       CALL #"LCP71_B010_BG8011"
       (
         CM_No       := 10174 ,
         Tab       := 1 ,
         SubTab       := 4 ,
         CfgType       := 0 ,
         CfgInvert       := True ,
         InputRaw       := LCP71_B010_BG8011_DI_ChA ,
         SC_Local       := SL_24_P ,
         CM_ALM        := "dbPlcHmiALM".ALM[10174] ,
       );

NETWORK
TITLE = 10175 - LCP71_B010_BG8012 - Door Hopper feeder Door - Safety Contact

       CALL #"LCP71_B010_BG8012"
       (
         CM_No       := 10175 ,
         Tab       := 1 ,
         SubTab       := 4 ,
         CfgType       := 0 ,
         CfgInvert       := True ,
         InputRaw       := LCP71_B010_BG8012_DI_ChA ,
         SC_Local       := SL_24_P ,
         CM_ALM        := "dbPlcHmiALM".ALM[10175] ,
       );

NETWORK
TITLE = 10176 - LCP71_B010_BG8013 - Hopper feeder Life Line  - Safety Contact

       CALL #"LCP71_B010_BG8013"
       (
         CM_No       := 10176 ,
         Tab       := 1 ,
         SubTab       := 4 ,
         CfgType       := 0 ,
         CfgInvert       := True ,
         InputRaw       := LCP71_B010_BG8013_DI_ChA ,
         SC_Local       := SL_24_P ,
         CM_ALM        := "dbPlcHmiALM".ALM[10176] ,
       );

NETWORK
TITLE = 10177 - LCP71_ES01_SF6134 - Emergency Stop  - Hopper Feeder

       CALL #"LCP71_ES01_SF6134"
       (
         CM_No       := 10177 ,
         Tab       := 1 ,
         SubTab       := 4 ,
         CfgType       := 0 ,
         CfgInvert       := True ,
         InputRaw       := LCP71_ES01_SF6134_DI_ChA ,
         SC_Local       := SL_01 ,
         CM_ALM        := "dbPlcHmiALM".ALM[10177] ,
       );

NETWORK
TITLE = 10178 - LCP71_ES01_SF6135 - Emergency Stop  - LCP71

       CALL #"LCP71_ES01_SF6135"
       (
         CM_No       := 10178 ,
         Tab       := 1 ,
         SubTab       := 4 ,
         CfgType       := 0 ,
         CfgInvert       := True ,
         InputRaw       := LCP71_ES01_SF6135_DI_ChA ,
         SC_Local       := SL_01 ,
         CM_ALM        := "dbPlcHmiALM".ALM[10178] ,
       );

NETWORK
TITLE = 10179 - LCP71_DC01_FC1000 - Power Feed Module 24VDC - Status

       CALL #"LCP71_DC01_FC1000"
       (
         CM_No       := 10179 ,
         Tab       := 13 ,
         SubTab       := 5 ,
         CfgType       := 0 ,
         CfgInvert       := True ,
         InputRaw       := LCP71_DC01_FC1000_DI_Sts ,
         SC_Local       := SL_13 ,
         CM_ALM        := "dbPlcHmiALM".ALM[10179] ,
       );

NETWORK
TITLE = 10180 - LCP71_IO_KF1000 - Point IO - EtherNet/IP Adapter

       CALL #"LCP71_IO_KF1000"
       (
         CM_No       := 10180 ,
         Tab       := 13 ,
         SubTab       := 5 ,
         CfgType       := 0 ,
         CfgInvert       := True ,
         InputRaw       :=  ,
         SC_Local       := SL_13 ,
         CM_ALM        := "dbPlcHmiALM".ALM[10180] ,
       );

NETWORK
TITLE = 10181 - LCP71_IO_KF3007 - 24V DC 8-Point Safety Input Module - SDI

       CALL #"LCP71_IO_KF3007"
       (
         CM_No       := 10181 ,
         Tab       := 13 ,
         SubTab       := 5 ,
         CfgType       := 0 ,
         CfgInvert       := True ,
         InputRaw       :=  ,
         SC_Local       := SL_13 ,
         CM_ALM        := "dbPlcHmiALM".ALM[10181] ,
       );

NETWORK
TITLE = 10182 - LCP71_IO_KF3008 - 24V DC 8-Point Safety Input Module - SDI

       CALL #"LCP71_IO_KF3008"
       (
         CM_No       := 10182 ,
         Tab       := 13 ,
         SubTab       := 5 ,
         CfgType       := 0 ,
         CfgInvert       := True ,
         InputRaw       :=  ,
         SC_Local       := SL_13 ,
         CM_ALM        := "dbPlcHmiALM".ALM[10182] ,
       );

NETWORK
TITLE = 10183 - LCP72_B211_BG8211 - Conderser 2 Door - Safety Contact

       CALL #"LCP72_B211_BG8211"
       (
         CM_No       := 10183 ,
         Tab       := 1 ,
         SubTab       := 4 ,
         CfgType       := 0 ,
         CfgInvert       := True ,
         InputRaw       := LCP72_B211_BG8211_DI_ChA ,
         SC_Local       := SL_24_P12 ,
         CM_ALM        := "dbPlcHmiALM".ALM[10183] ,
       );

NETWORK
TITLE = 10184 - LCP72_B311_BG8311 - Conderser 3 Door - Safety Contact

       CALL #"LCP72_B311_BG8311"
       (
         CM_No       := 10184 ,
         Tab       := 1 ,
         SubTab       := 4 ,
         CfgType       := 0 ,
         CfgInvert       := True ,
         InputRaw       := LCP72_B311_BG8311_DI_ChA ,
         SC_Local       := SL_24_P13 ,
         CM_ALM        := "dbPlcHmiALM".ALM[10184] ,
       );

NETWORK
TITLE = 10185 - LCP72_B411_BG8411 - Conderser 4 Door - Safety Contact

       CALL #"LCP72_B411_BG8411"
       (
         CM_No       := 10185 ,
         Tab       := 1 ,
         SubTab       := 4 ,
         CfgType       := 0 ,
         CfgInvert       := True ,
         InputRaw       := LCP72_B411_BG8411_DI_ChA ,
         SC_Local       := SL_24_P14 ,
         CM_ALM        := "dbPlcHmiALM".ALM[10185] ,
       );

NETWORK
TITLE = 10186 - LCP72_B210_KF6210 - Opening Roll 2 Rotation Monitor - Fault

       CALL #"LCP72_B210_KF6210"
       (
         CM_No       := 10186 ,
         Tab       := 24 ,
         SubTab       := 4 ,
         CfgType       := 0 ,
         CfgInvert       := True ,
         InputRaw       := LCP72_B210_KF6210_DI_Flt ,
         SC_Local       := SL_24_P12 ,
         CM_ALM        := "dbPlcHmiALM".ALM[10186] ,
       );

NETWORK
TITLE = 10187 - LCP72_B210_RL4210 - Metering Feeder 2 - Door Lock Open

       CALL #"LCP72_B210_RL4210"
       (
         CM_No       := 10187 ,
         Tab       := 1 ,
         SubTab       := 4 ,
         CfgType       := 0 ,
         CfgInvert       := True ,
         InputRaw       := LCP72_B210_RL4210_DI_ChA ,
         SC_Local       := SL_24_P12 ,
         CM_ALM        := "dbPlcHmiALM".ALM[10187] ,
       );

NETWORK
TITLE = 10188 - LCP72_B310_KF6310 - Opening Roll 3 Rotation Monitor - Fault

       CALL #"LCP72_B310_KF6310"
       (
         CM_No       := 10188 ,
         Tab       := 24 ,
         SubTab       := 5 ,
         CfgType       := 0 ,
         CfgInvert       := True ,
         InputRaw       := LCP72_B310_KF6310_DI_Flt ,
         SC_Local       := SL_24_P13 ,
         CM_ALM        := "dbPlcHmiALM".ALM[10188] ,
       );

NETWORK
TITLE = 10189 - LCP72_B310_RL4310 - Metering Feeder 3 - Door Lock Open

       CALL #"LCP72_B310_RL4310"
       (
         CM_No       := 10189 ,
         Tab       := 1 ,
         SubTab       := 4 ,
         CfgType       := 0 ,
         CfgInvert       := True ,
         InputRaw       := LCP72_B310_RL4310_DI_ChA ,
         SC_Local       := SL_24_P13 ,
         CM_ALM        := "dbPlcHmiALM".ALM[10189] ,
       );

NETWORK
TITLE = 10190 - LCP72_B410_KF6410 - Opening Roll 4 Rotation Monitor - Fault

       CALL #"LCP72_B410_KF6410"
       (
         CM_No       := 10190 ,
         Tab       := 24 ,
         SubTab       := 6 ,
         CfgType       := 0 ,
         CfgInvert       := True ,
         InputRaw       := LCP72_B410_KF6410_DI_Flt ,
         SC_Local       := SL_24_P14 ,
         CM_ALM        := "dbPlcHmiALM".ALM[10190] ,
       );

NETWORK
TITLE = 10191 - LCP72_B410_RL4410 - Metering Feeder 4 - Door Lock Open

       CALL #"LCP72_B410_RL4410"
       (
         CM_No       := 10191 ,
         Tab       := 1 ,
         SubTab       := 4 ,
         CfgType       := 0 ,
         CfgInvert       := True ,
         InputRaw       := LCP72_B410_RL4410_DI_ChA ,
         SC_Local       := SL_24_P14 ,
         CM_ALM        := "dbPlcHmiALM".ALM[10191] ,
       );

NETWORK
TITLE = 10192 - LCP72_B210_QA1201 - Serel 2 DCM - X-Ray Fault

       CALL #"LCP72_B210_QA1201"
       (
         CM_No       := 10192 ,
         Tab       := 24 ,
         SubTab       := 4 ,
         CfgType       := 0 ,
         CfgInvert       := True ,
         InputRaw       := LCP72_B210_QA1201_DI_Flt ,
         SC_Local       := SL_24_S ,
         CM_ALM        := "dbPlcHmiALM".ALM[10192] ,
       );

NETWORK
TITLE = 10193 - LCP72_B310_QA1301 - Serel 3 DCM - X-Ray Fault

       CALL #"LCP72_B310_QA1301"
       (
         CM_No       := 10193 ,
         Tab       := 24 ,
         SubTab       := 5 ,
         CfgType       := 0 ,
         CfgInvert       := True ,
         InputRaw       := LCP72_B310_QA1301_DI_Flt ,
         SC_Local       := SL_24_S ,
         CM_ALM        := "dbPlcHmiALM".ALM[10193] ,
       );

NETWORK
TITLE = 10194 - LCP72_B410_QA1401 - Serel 4 DCM - X-Ray Fault

       CALL #"LCP72_B410_QA1401"
       (
         CM_No       := 10194 ,
         Tab       := 24 ,
         SubTab       := 6 ,
         CfgType       := 0 ,
         CfgInvert       := True ,
         InputRaw       := LCP72_B410_QA1401_DI_Flt ,
         SC_Local       := SL_24_S ,
         CM_ALM        := "dbPlcHmiALM".ALM[10194] ,
       );

NETWORK
TITLE = 10195 - LCP72_ES01_SF6130 - Emergency Stop  - Meeting Feeder 1

       CALL #"LCP72_ES01_SF6130"
       (
         CM_No       := 10195 ,
         Tab       := 1 ,
         SubTab       := 4 ,
         CfgType       := 0 ,
         CfgInvert       := True ,
         InputRaw       := LCP72_ES01_SF6130_DI_ChA ,
         SC_Local       := SL_01 ,
         CM_ALM        := "dbPlcHmiALM".ALM[10195] ,
       );

NETWORK
TITLE = 10196 - LCP72_ES01_SF6131 - Emergency Stop  - Meeting Feeder 2

       CALL #"LCP72_ES01_SF6131"
       (
         CM_No       := 10196 ,
         Tab       := 1 ,
         SubTab       := 4 ,
         CfgType       := 0 ,
         CfgInvert       := True ,
         InputRaw       := LCP72_ES01_SF6131_DI_ChA ,
         SC_Local       := SL_01 ,
         CM_ALM        := "dbPlcHmiALM".ALM[10196] ,
       );

NETWORK
TITLE = 10197 - LCP72_ES01_SF6132 - Emergency Stop  - Meeting Feeder 3

       CALL #"LCP72_ES01_SF6132"
       (
         CM_No       := 10197 ,
         Tab       := 1 ,
         SubTab       := 4 ,
         CfgType       := 0 ,
         CfgInvert       := True ,
         InputRaw       := LCP72_ES01_SF6132_DI_ChA ,
         SC_Local       := SL_01 ,
         CM_ALM        := "dbPlcHmiALM".ALM[10197] ,
       );

NETWORK
TITLE = 10198 - LCP72_ES01_SF6133 - Emergency Stop  - LCP72

       CALL #"LCP72_ES01_SF6133"
       (
         CM_No       := 10198 ,
         Tab       := 1 ,
         SubTab       := 4 ,
         CfgType       := 0 ,
         CfgInvert       := True ,
         InputRaw       := LCP72_ES01_SF6133_DI_ChA ,
         SC_Local       := SL_01 ,
         CM_ALM        := "dbPlcHmiALM".ALM[10198] ,
       );

NETWORK
TITLE = 10199 - LCP72_DC01_FC1000 - Power Feed Module 24VDC - Status

       CALL #"LCP72_DC01_FC1000"
       (
         CM_No       := 10199 ,
         Tab       := 13 ,
         SubTab       := 5 ,
         CfgType       := 0 ,
         CfgInvert       := True ,
         InputRaw       := LCP72_DC01_FC1000_DI_Sts ,
         SC_Local       := SL_13 ,
         CM_ALM        := "dbPlcHmiALM".ALM[10199] ,
       );

NETWORK
TITLE = 10200 - LCP72_IO_KF1000 - Point IO - EtherNet/IP Adapter

       CALL #"LCP72_IO_KF1000"
       (
         CM_No       := 10200 ,
         Tab       := 13 ,
         SubTab       := 5 ,
         CfgType       := 0 ,
         CfgInvert       := True ,
         InputRaw       :=  ,
         SC_Local       := SL_13 ,
         CM_ALM        := "dbPlcHmiALM".ALM[10200] ,
       );

NETWORK
TITLE = 10201 - LCP72_IO_KF3017 - 24V DC 8-Point Safety Input Module - SDI

       CALL #"LCP72_IO_KF3017"
       (
         CM_No       := 10201 ,
         Tab       := 13 ,
         SubTab       := 5 ,
         CfgType       := 0 ,
         CfgInvert       := True ,
         InputRaw       :=  ,
         SC_Local       := SL_13 ,
         CM_ALM        := "dbPlcHmiALM".ALM[10201] ,
       );

NETWORK
TITLE = 10202 - LCP72_IO_KF3018 - 24V DC 8-Point Safety Input Module - SDI

       CALL #"LCP72_IO_KF3018"
       (
         CM_No       := 10202 ,
         Tab       := 13 ,
         SubTab       := 5 ,
         CfgType       := 0 ,
         CfgInvert       := True ,
         InputRaw       :=  ,
         SC_Local       := SL_13 ,
         CM_ALM        := "dbPlcHmiALM".ALM[10202] ,
       );

NETWORK
TITLE = 10203 - LCP72_IO_KF3019 - 24V DC 8-Point Safety Input Module - SDI

       CALL #"LCP72_IO_KF3019"
       (
         CM_No       := 10203 ,
         Tab       := 13 ,
         SubTab       := 5 ,
         CfgType       := 0 ,
         CfgInvert       := True ,
         InputRaw       :=  ,
         SC_Local       := SL_13 ,
         CM_ALM        := "dbPlcHmiALM".ALM[10203] ,
       );

NETWORK
TITLE = 10204 - LCP72_IO_KF3020 - 24V DC 8-Point Safety Input Module - SDI

       CALL #"LCP72_IO_KF3020"
       (
         CM_No       := 10204 ,
         Tab       := 13 ,
         SubTab       := 5 ,
         CfgType       := 0 ,
         CfgInvert       := True ,
         InputRaw       :=  ,
         SC_Local       := SL_13 ,
         CM_ALM        := "dbPlcHmiALM".ALM[10204] ,
       );

NETWORK
TITLE = 10205 - LCP72_IO_KF3021 - 24V DC 8-Point Source Safety Output Module - SDO

       CALL #"LCP72_IO_KF3021"
       (
         CM_No       := 10205 ,
         Tab       := 13 ,
         SubTab       := 5 ,
         CfgType       := 0 ,
         CfgInvert       := True ,
         InputRaw       :=  ,
         SC_Local       := SL_13 ,
         CM_ALM        := "dbPlcHmiALM".ALM[10205] ,
       );

NETWORK
TITLE = 10206 - LCP81_C311_BG6311 - Compactor Up Pos. OS - Up

       CALL #"LCP81_C311_BG6311"
       (
         CM_No       := 10206 ,
         Tab       := 26 ,
         SubTab       := 7 ,
         CfgType       := 0 ,
         CfgInvert       := True ,
         InputRaw       := LCP81_C311_BG6311_DI_FbP ,
         SC_Local       := SL_26_P ,
         CM_ALM        := "dbPlcHmiALM".ALM[10206] ,
       );

NETWORK
TITLE = 10207 - LCP81_C311_BG6312 - Compactor Up Pos. DS - Up

       CALL #"LCP81_C311_BG6312"
       (
         CM_No       := 10207 ,
         Tab       := 26 ,
         SubTab       := 7 ,
         CfgType       := 0 ,
         CfgInvert       := True ,
         InputRaw       := LCP81_C311_BG6312_DI_FbP ,
         SC_Local       := SL_26_P ,
         CM_ALM        := "dbPlcHmiALM".ALM[10207] ,
       );

NETWORK
TITLE = 10208 - LCP81_C311_BG6313 - Compactor after Lock Pos. - Read Contact

       CALL #"LCP81_C311_BG6313"
       (
         CM_No       := 10208 ,
         Tab       := 26 ,
         SubTab       := 7 ,
         CfgType       := 0 ,
         CfgInvert       := True ,
         InputRaw       := LCP81_C311_BG6313_DI_FbAl ,
         SC_Local       := SL_26_P ,
         CM_ALM        := "dbPlcHmiALM".ALM[10208] ,
       );

NETWORK
TITLE = 10209 - LCP81_C311_BG6314 - Compactor Lock In Pos. OS - Locked

       CALL #"LCP81_C311_BG6314"
       (
         CM_No       := 10209 ,
         Tab       := 26 ,
         SubTab       := 7 ,
         CfgType       := 0 ,
         CfgInvert       := True ,
         InputRaw       := LCP81_C311_BG6314_DI_FbP ,
         SC_Local       := SL_26_P ,
         CM_ALM        := "dbPlcHmiALM".ALM[10209] ,
       );

NETWORK
TITLE = 10210 - LCP81_C311_BG6315 - Compactor Lock Out Pos. OS - Unlocked

       CALL #"LCP81_C311_BG6315"
       (
         CM_No       := 10210 ,
         Tab       := 26 ,
         SubTab       := 7 ,
         CfgType       := 0 ,
         CfgInvert       := True ,
         InputRaw       := LCP81_C311_BG6315_DI_FbN ,
         SC_Local       := SL_26_P ,
         CM_ALM        := "dbPlcHmiALM".ALM[10210] ,
       );

NETWORK
TITLE = 10211 - LCP81_C311_BG6316 - Compactor Lock In Pos. DS - Locked

       CALL #"LCP81_C311_BG6316"
       (
         CM_No       := 10211 ,
         Tab       := 26 ,
         SubTab       := 7 ,
         CfgType       := 0 ,
         CfgInvert       := True ,
         InputRaw       := LCP81_C311_BG6316_DI_FbP ,
         SC_Local       := SL_26_P ,
         CM_ALM        := "dbPlcHmiALM".ALM[10211] ,
       );

NETWORK
TITLE = 10212 - LCP81_C311_BG6317 - Compactor Lock Out Pos. DS - Unlocked

       CALL #"LCP81_C311_BG6317"
       (
         CM_No       := 10212 ,
         Tab       := 26 ,
         SubTab       := 7 ,
         CfgType       := 0 ,
         CfgInvert       := True ,
         InputRaw       := LCP81_C311_BG6317_DI_FbN ,
         SC_Local       := SL_26_P ,
         CM_ALM        := "dbPlcHmiALM".ALM[10212] ,
       );

NETWORK
TITLE = 10213 - LCP81_ES01_SF6136 - Emergency Stop  - Dryer 1 Ratio Box CB.81-01

       CALL #"LCP81_ES01_SF6136"
       (
         CM_No       := 10213 ,
         Tab       := 1 ,
         SubTab       := 5 ,
         CfgType       := 0 ,
         CfgInvert       := True ,
         InputRaw       := LCP81_ES01_SF6136_DI_ChA ,
         SC_Local       := SL_01 ,
         CM_ALM        := "dbPlcHmiALM".ALM[10213] ,
       );

NETWORK
TITLE = 10214 - LCP81_ES01_SF6137 - Emergency Stop  - Former Fan area

       CALL #"LCP81_ES01_SF6137"
       (
         CM_No       := 10214 ,
         Tab       := 1 ,
         SubTab       := 5 ,
         CfgType       := 0 ,
         CfgInvert       := True ,
         InputRaw       := LCP81_ES01_SF6137_DI_ChA ,
         SC_Local       := SL_01 ,
         CM_ALM        := "dbPlcHmiALM".ALM[10214] ,
       );

NETWORK
TITLE = 10215 - LCP81_ES01_SF6138 - Emergency Stop  - Former Fan area

       CALL #"LCP81_ES01_SF6138"
       (
         CM_No       := 10215 ,
         Tab       := 1 ,
         SubTab       := 5 ,
         CfgType       := 0 ,
         CfgInvert       := True ,
         InputRaw       := LCP81_ES01_SF6138_DI_ChA ,
         SC_Local       := SL_01 ,
         CM_ALM        := "dbPlcHmiALM".ALM[10215] ,
       );

NETWORK
TITLE = 10216 - LCP81_ES01_SF6139 - Emergency Stop  - LCP81

       CALL #"LCP81_ES01_SF6139"
       (
         CM_No       := 10216 ,
         Tab       := 1 ,
         SubTab       := 5 ,
         CfgType       := 0 ,
         CfgInvert       := True ,
         InputRaw       := LCP81_ES01_SF6139_DI_ChA ,
         SC_Local       := SL_01 ,
         CM_ALM        := "dbPlcHmiALM".ALM[10216] ,
       );

NETWORK
TITLE = 10217 - LCP81_DC01_FC1000 - Power Feed Module 24VDC - Status

       CALL #"LCP81_DC01_FC1000"
       (
         CM_No       := 10217 ,
         Tab       := 13 ,
         SubTab       := 5 ,
         CfgType       := 0 ,
         CfgInvert       := True ,
         InputRaw       := LCP81_DC01_FC1000_DI_Sts ,
         SC_Local       := SL_13 ,
         CM_ALM        := "dbPlcHmiALM".ALM[10217] ,
       );

NETWORK
TITLE = 10218 - LCP81_IO_KF1000 - Point IO - EtherNet/IP Adapter

       CALL #"LCP81_IO_KF1000"
       (
         CM_No       := 10218 ,
         Tab       := 13 ,
         SubTab       := 5 ,
         CfgType       := 0 ,
         CfgInvert       := True ,
         InputRaw       :=  ,
         SC_Local       := SL_13 ,
         CM_ALM        := "dbPlcHmiALM".ALM[10218] ,
       );

NETWORK
TITLE = 10219 - LCP81_IO_KF2000 - Point IO 2nd - EtherNet/IP Adapter

       CALL #"LCP81_IO_KF2000"
       (
         CM_No       := 10219 ,
         Tab       := 13 ,
         SubTab       := 5 ,
         CfgType       := 0 ,
         CfgInvert       := True ,
         InputRaw       :=  ,
         SC_Local       := SL_13 ,
         CM_ALM        := "dbPlcHmiALM".ALM[10219] ,
       );

NETWORK
TITLE = 10220 - LCP81_IO_KF3047 - 24V DC 8-Point Safety Input Module - SDI

       CALL #"LCP81_IO_KF3047"
       (
         CM_No       := 10220 ,
         Tab       := 13 ,
         SubTab       := 5 ,
         CfgType       := 0 ,
         CfgInvert       := True ,
         InputRaw       :=  ,
         SC_Local       := SL_13 ,
         CM_ALM        := "dbPlcHmiALM".ALM[10220] ,
       );

NETWORK
TITLE = 10221 - LCP81_IO_KF3048 - 24V DC 8-Point Safety Input Module - SDI

       CALL #"LCP81_IO_KF3048"
       (
         CM_No       := 10221 ,
         Tab       := 13 ,
         SubTab       := 5 ,
         CfgType       := 0 ,
         CfgInvert       := True ,
         InputRaw       :=  ,
         SC_Local       := SL_13 ,
         CM_ALM        := "dbPlcHmiALM".ALM[10221] ,
       );

NETWORK
TITLE = 10222 - LCP91_A110_SF6141 - Filter 1 Zone 1 - Ex doors & Estop

       CALL #"LCP91_A110_SF6141"
       (
         CM_No       := 10222 ,
         Tab       := 1 ,
         SubTab       := 3 ,
         CfgType       := 0 ,
         CfgInvert       := True ,
         InputRaw       := LCP91_A110_SF6141_DI_ChA ,
         SC_Local       := SL_01 ,
         CM_ALM        := "dbPlcHmiALM".ALM[10222] ,
       );

NETWORK
TITLE = 10223 - LCP91_A110_BG7712 - Filter 1 Zone 2 - Top Door

       CALL #"LCP91_A110_BG7712"
       (
         CM_No       := 10223 ,
         Tab       := 1 ,
         SubTab       := 3 ,
         CfgType       := 0 ,
         CfgInvert       := True ,
         InputRaw       := LCP91_A110_BG7712_DI_ChA ,
         SC_Local       := SL_01 ,
         CM_ALM        := "dbPlcHmiALM".ALM[10223] ,
       );

NETWORK
TITLE = 10224 - LCP91_A110_BG7711 - Filter 1 Zone 3 - Bottom Doors

       CALL #"LCP91_A110_BG7711"
       (
         CM_No       := 10224 ,
         Tab       := 1 ,
         SubTab       := 3 ,
         CfgType       := 0 ,
         CfgInvert       := True ,
         InputRaw       := LCP91_A110_BG7711_DI_ChA ,
         SC_Local       := SL_01 ,
         CM_ALM        := "dbPlcHmiALM".ALM[10224] ,
       );

NETWORK
TITLE = 10225 - LCP91_ES01_SF6142 - Emergency Stop  - LCP91

       CALL #"LCP91_ES01_SF6142"
       (
         CM_No       := 10225 ,
         Tab       := 1 ,
         SubTab       := 3 ,
         CfgType       := 0 ,
         CfgInvert       := True ,
         InputRaw       := LCP91_ES01_SF6142_DI_ChA ,
         SC_Local       := SL_01 ,
         CM_ALM        := "dbPlcHmiALM".ALM[10225] ,
       );

NETWORK
TITLE = 10226 - LCP91_DC01_FC1000 - Power Feed Module 24VDC - Status

       CALL #"LCP91_DC01_FC1000"
       (
         CM_No       := 10226 ,
         Tab       := 13 ,
         SubTab       := 5 ,
         CfgType       := 0 ,
         CfgInvert       := True ,
         InputRaw       := LCP91_DC01_FC1000_DI_Sts ,
         SC_Local       := SL_13 ,
         CM_ALM        := "dbPlcHmiALM".ALM[10226] ,
       );

NETWORK
TITLE = 10227 - LCP91_IO_KF1000 - Point IO - EtherNet/IP Adapter

       CALL #"LCP91_IO_KF1000"
       (
         CM_No       := 10227 ,
         Tab       := 13 ,
         SubTab       := 5 ,
         CfgType       := 0 ,
         CfgInvert       := True ,
         InputRaw       :=  ,
         SC_Local       := SL_13 ,
         CM_ALM        := "dbPlcHmiALM".ALM[10227] ,
       );

NETWORK
TITLE = 10228 - LCP91_IO_KF3015 - 24V DC 8-Point Safety Input Module - SDI

       CALL #"LCP91_IO_KF3015"
       (
         CM_No       := 10228 ,
         Tab       := 13 ,
         SubTab       := 5 ,
         CfgType       := 0 ,
         CfgInvert       := True ,
         InputRaw       :=  ,
         SC_Local       := SL_13 ,
         CM_ALM        := "dbPlcHmiALM".ALM[10228] ,
       );

NETWORK
TITLE = 10229 - LCP91_IO_KF3016 - 24V DC 8-Point Safety Input Module - SDI

       CALL #"LCP91_IO_KF3016"
       (
         CM_No       := 10229 ,
         Tab       := 13 ,
         SubTab       := 5 ,
         CfgType       := 0 ,
         CfgInvert       := True ,
         InputRaw       :=  ,
         SC_Local       := SL_13 ,
         CM_ALM        := "dbPlcHmiALM".ALM[10229] ,
       );

NETWORK
TITLE = 10230 - LCP91_IO_KF3017 - 24V DC IO Link Master Module - IO Link

       CALL #"LCP91_IO_KF3017"
       (
         CM_No       := 10230 ,
         Tab       := 13 ,
         SubTab       := 5 ,
         CfgType       := 0 ,
         CfgInvert       := True ,
         InputRaw       :=  ,
         SC_Local       := SL_13 ,
         CM_ALM        := "dbPlcHmiALM".ALM[10230] ,
       );

NETWORK
TITLE = 10231 - LCP92_A210_CB.A210-14 - Control Box - Baghouse Filter 2

       CALL #"LCP92_A210_CB.A210-14"
       (
         CM_No       := 10231 ,
         Tab       := 21 ,
         SubTab       := 2 ,
         CfgType       := 0 ,
         CfgInvert       := True ,
         InputRaw       :=  ,
         SC_Local       := SL_01 ,
         CM_ALM        := "dbPlcHmiALM".ALM[10231] ,
       );

NETWORK
TITLE = 10232 - LCP92_A210_SF6144 - Filter 2 Zone 1 - Ex doors & Estop

       CALL #"LCP92_A210_SF6144"
       (
         CM_No       := 10232 ,
         Tab       := 1 ,
         SubTab       := 3 ,
         CfgType       := 0 ,
         CfgInvert       := True ,
         InputRaw       := LCP92_A210_SF6144_DI_ChA ,
         SC_Local       := SL_01 ,
         CM_ALM        := "dbPlcHmiALM".ALM[10232] ,
       );

NETWORK
TITLE = 10233 - LCP92_A210_CB.A210-15 - Control Box - Baghouse Filter 2

       CALL #"LCP92_A210_CB.A210-15"
       (
         CM_No       := 10233 ,
         Tab       := 21 ,
         SubTab       := 2 ,
         CfgType       := 0 ,
         CfgInvert       := True ,
         InputRaw       :=  ,
         SC_Local       := SL_01 ,
         CM_ALM        := "dbPlcHmiALM".ALM[10233] ,
       );

NETWORK
TITLE = 10234 - LCP92_A210_BG7732 - Filter 2 Zone 2 - Top Door

       CALL #"LCP92_A210_BG7732"
       (
         CM_No       := 10234 ,
         Tab       := 1 ,
         SubTab       := 3 ,
         CfgType       := 0 ,
         CfgInvert       := True ,
         InputRaw       := LCP92_A210_BG7732_DI_ChA ,
         SC_Local       := SL_01 ,
         CM_ALM        := "dbPlcHmiALM".ALM[10234] ,
       );

NETWORK
TITLE = 10235 - LCP92_A210_BG7731 - Filter 2 Zone 3 - Bottom Doors

       CALL #"LCP92_A210_BG7731"
       (
         CM_No       := 10235 ,
         Tab       := 1 ,
         SubTab       := 3 ,
         CfgType       := 0 ,
         CfgInvert       := True ,
         InputRaw       := LCP92_A210_BG7731_DI_ChA ,
         SC_Local       := SL_01 ,
         CM_ALM        := "dbPlcHmiALM".ALM[10235] ,
       );

NETWORK
TITLE = 10236 - LCP92_ES01_SF6145 - Emergency Stop  - LCP92

       CALL #"LCP92_ES01_SF6145"
       (
         CM_No       := 10236 ,
         Tab       := 1 ,
         SubTab       := 3 ,
         CfgType       := 0 ,
         CfgInvert       := True ,
         InputRaw       := LCP92_ES01_SF6145_DI_ChA ,
         SC_Local       := SL_01 ,
         CM_ALM        := "dbPlcHmiALM".ALM[10236] ,
       );

NETWORK
TITLE = 10237 - LCP92_DC01_FC1000 - Power Feed Module 24VDC - Status

       CALL #"LCP92_DC01_FC1000"
       (
         CM_No       := 10237 ,
         Tab       := 13 ,
         SubTab       := 5 ,
         CfgType       := 0 ,
         CfgInvert       := True ,
         InputRaw       := LCP92_DC01_FC1000_DI_Flt ,
         SC_Local       := SL_13 ,
         CM_ALM        := "dbPlcHmiALM".ALM[10237] ,
       );

NETWORK
TITLE = 10238 - LCP92_IO_KF1000 - Point IO - EtherNet/IP Adapter

       CALL #"LCP92_IO_KF1000"
       (
         CM_No       := 10238 ,
         Tab       := 13 ,
         SubTab       := 5 ,
         CfgType       := 0 ,
         CfgInvert       := True ,
         InputRaw       :=  ,
         SC_Local       := SL_13 ,
         CM_ALM        := "dbPlcHmiALM".ALM[10238] ,
       );

NETWORK
TITLE = 10239 - LCP92_IO_KF3013 - 24V DC 8-Point Safety Input Module - SDI

       CALL #"LCP92_IO_KF3013"
       (
         CM_No       := 10239 ,
         Tab       := 13 ,
         SubTab       := 5 ,
         CfgType       := 0 ,
         CfgInvert       := True ,
         InputRaw       :=  ,
         SC_Local       := SL_13 ,
         CM_ALM        := "dbPlcHmiALM".ALM[10239] ,
       );

NETWORK
TITLE = 10240 - LCP92_IO_KF3014 - 24V DC 8-Point Safety Input Module - SDI

       CALL #"LCP92_IO_KF3014"
       (
         CM_No       := 10240 ,
         Tab       := 13 ,
         SubTab       := 5 ,
         CfgType       := 0 ,
         CfgInvert       := True ,
         InputRaw       :=  ,
         SC_Local       := SL_13 ,
         CM_ALM        := "dbPlcHmiALM".ALM[10240] ,
       );

NETWORK
TITLE = 10241 - LCP92_IO_KF3015 - 24V DC IO Link Master Module - IO Link

       CALL #"LCP92_IO_KF3015"
       (
         CM_No       := 10241 ,
         Tab       := 13 ,
         SubTab       := 5 ,
         CfgType       := 0 ,
         CfgInvert       := True ,
         InputRaw       :=  ,
         SC_Local       := SL_13 ,
         CM_ALM        := "dbPlcHmiALM".ALM[10241] ,
       );

NETWORK
TITLE = 10242 - LCP93_A171_FN3771 - Humidifier 1 Fan 1  - Motor Disconnect

       CALL #"LCP93_A171_FN3771"
       (
         CM_No       := 10242 ,
         Tab       := 22 ,
         SubTab       := 4 ,
         CfgType       := 0 ,
         CfgInvert       := True ,
         InputRaw       := LCP93_A171_FN3771_DI_Flt ,
         SC_Local       := SL_22_P ,
         CM_ALM        := "dbPlcHmiALM".ALM[10242] ,
       );

NETWORK
TITLE = 10243 - LCP93_A172_FN3772 - Humidifier 1 Fan 2  - Motor Disconnect

       CALL #"LCP93_A172_FN3772"
       (
         CM_No       := 10243 ,
         Tab       := 22 ,
         SubTab       := 4 ,
         CfgType       := 0 ,
         CfgInvert       := True ,
         InputRaw       := LCP93_A172_FN3772_DI_Flt ,
         SC_Local       := SL_22_P ,
         CM_ALM        := "dbPlcHmiALM".ALM[10243] ,
       );

NETWORK
TITLE = 10244 - LCP93_A173_FN3773 - Humidifier 1 Fan 3  - Motor Disconnect

       CALL #"LCP93_A173_FN3773"
       (
         CM_No       := 10244 ,
         Tab       := 22 ,
         SubTab       := 4 ,
         CfgType       := 0 ,
         CfgInvert       := True ,
         InputRaw       := LCP93_A173_FN3773_DI_Flt ,
         SC_Local       := SL_22_P ,
         CM_ALM        := "dbPlcHmiALM".ALM[10244] ,
       );

NETWORK
TITLE = 10245 - LCP93_A174_FN3774 - Humidifier 1 Fan 4  - Motor Disconnect

       CALL #"LCP93_A174_FN3774"
       (
         CM_No       := 10245 ,
         Tab       := 22 ,
         SubTab       := 4 ,
         CfgType       := 0 ,
         CfgInvert       := True ,
         InputRaw       := LCP93_A174_FN3774_DI_Flt ,
         SC_Local       := SL_22_P ,
         CM_ALM        := "dbPlcHmiALM".ALM[10245] ,
       );

NETWORK
TITLE = 10246 - LCP93_A191_FN3781 - Humidifier 3 Fan 1  - Motor Disconnect

       CALL #"LCP93_A191_FN3781"
       (
         CM_No       := 10246 ,
         Tab       := 22 ,
         SubTab       := 5 ,
         CfgType       := 0 ,
         CfgInvert       := True ,
         InputRaw       := LCP93_A191_FN3781_DI_Flt ,
         SC_Local       := SL_22_P ,
         CM_ALM        := "dbPlcHmiALM".ALM[10246] ,
       );

NETWORK
TITLE = 10247 - LCP93_A192_FN3782 - Humidifier 3 Fan 2  - Motor Disconnect

       CALL #"LCP93_A192_FN3782"
       (
         CM_No       := 10247 ,
         Tab       := 22 ,
         SubTab       := 5 ,
         CfgType       := 0 ,
         CfgInvert       := True ,
         InputRaw       := LCP93_A192_FN3782_DI_Flt ,
         SC_Local       := SL_22_P ,
         CM_ALM        := "dbPlcHmiALM".ALM[10247] ,
       );

NETWORK
TITLE = 10248 - LCP93_A193_FN3783 - Humidifier 3 Fan 3 - Motor Disconnect

       CALL #"LCP93_A193_FN3783"
       (
         CM_No       := 10248 ,
         Tab       := 22 ,
         SubTab       := 5 ,
         CfgType       := 0 ,
         CfgInvert       := True ,
         InputRaw       := LCP93_A193_FN3783_DI_Flt ,
         SC_Local       := SL_22_P ,
         CM_ALM        := "dbPlcHmiALM".ALM[10248] ,
       );

NETWORK
TITLE = 10249 - LCP93_A194_FN3784 - Humidifier 3 Fan 4 - Motor Disconnect

       CALL #"LCP93_A194_FN3784"
       (
         CM_No       := 10249 ,
         Tab       := 22 ,
         SubTab       := 5 ,
         CfgType       := 0 ,
         CfgInvert       := True ,
         InputRaw       := LCP93_A194_FN3784_DI_Flt ,
         SC_Local       := SL_22_P ,
         CM_ALM        := "dbPlcHmiALM".ALM[10249] ,
       );

NETWORK
TITLE = 10250 - LCP93_A271_FN3786 - Humidifier 4 Fan 1  - Motor Disconnect

       CALL #"LCP93_A271_FN3786"
       (
         CM_No       := 10250 ,
         Tab       := 22 ,
         SubTab       := 5 ,
         CfgType       := 0 ,
         CfgInvert       := True ,
         InputRaw       := LCP93_A271_FN3786_DI_Flt ,
         SC_Local       := SL_22_P ,
         CM_ALM        := "dbPlcHmiALM".ALM[10250] ,
       );

NETWORK
TITLE = 10251 - LCP93_A272_FN3787 - Humidifier 4 Fan 2  - Motor Disconnect

       CALL #"LCP93_A272_FN3787"
       (
         CM_No       := 10251 ,
         Tab       := 22 ,
         SubTab       := 5 ,
         CfgType       := 0 ,
         CfgInvert       := True ,
         InputRaw       := LCP93_A272_FN3787_DI_Flt ,
         SC_Local       := SL_22_P ,
         CM_ALM        := "dbPlcHmiALM".ALM[10251] ,
       );

NETWORK
TITLE = 10252 - LCP93_A273_FN3788 - Humidifier 4 Fan 3  - Motor Disconnect

       CALL #"LCP93_A273_FN3788"
       (
         CM_No       := 10252 ,
         Tab       := 22 ,
         SubTab       := 5 ,
         CfgType       := 0 ,
         CfgInvert       := True ,
         InputRaw       := LCP93_A273_FN3788_DI_Flt ,
         SC_Local       := SL_22_P ,
         CM_ALM        := "dbPlcHmiALM".ALM[10252] ,
       );

NETWORK
TITLE = 10253 - LCP93_A274_FN3789 - Humidifier 4 Fan 4 - Motor Disconnect

       CALL #"LCP93_A274_FN3789"
       (
         CM_No       := 10253 ,
         Tab       := 22 ,
         SubTab       := 5 ,
         CfgType       := 0 ,
         CfgInvert       := True ,
         InputRaw       := LCP93_A274_FN3789_DI_Flt ,
         SC_Local       := SL_22_P ,
         CM_ALM        := "dbPlcHmiALM".ALM[10253] ,
       );

NETWORK
TITLE = 10254 - LCP93_A281_FN3791 - Humidifier 5 Fan 1  - Motor Disconnect

       CALL #"LCP93_A281_FN3791"
       (
         CM_No       := 10254 ,
         Tab       := 22 ,
         SubTab       := 6 ,
         CfgType       := 0 ,
         CfgInvert       := True ,
         InputRaw       := LCP93_A281_FN3791_DI_Flt ,
         SC_Local       := SL_22_P ,
         CM_ALM        := "dbPlcHmiALM".ALM[10254] ,
       );

NETWORK
TITLE = 10255 - LCP93_A282_FN3792 - Humidifier 5 Fan 2  - Motor Disconnect

       CALL #"LCP93_A282_FN3792"
       (
         CM_No       := 10255 ,
         Tab       := 22 ,
         SubTab       := 6 ,
         CfgType       := 0 ,
         CfgInvert       := True ,
         InputRaw       := LCP93_A282_FN3792_DI_Flt ,
         SC_Local       := SL_22_P ,
         CM_ALM        := "dbPlcHmiALM".ALM[10255] ,
       );

NETWORK
TITLE = 10256 - LCP93_A283_FN3793 - Humidifier 5 Fan 3  - Motor Disconnect

       CALL #"LCP93_A283_FN3793"
       (
         CM_No       := 10256 ,
         Tab       := 22 ,
         SubTab       := 6 ,
         CfgType       := 0 ,
         CfgInvert       := True ,
         InputRaw       := LCP93_A283_FN3793_DI_Flt ,
         SC_Local       := SL_22_P ,
         CM_ALM        := "dbPlcHmiALM".ALM[10256] ,
       );

NETWORK
TITLE = 10257 - LCP93_A284_FN3794 - Humidifier 5 Fan 4  - Motor Disconnect

       CALL #"LCP93_A284_FN3794"
       (
         CM_No       := 10257 ,
         Tab       := 22 ,
         SubTab       := 6 ,
         CfgType       := 0 ,
         CfgInvert       := True ,
         InputRaw       := LCP93_A284_FN3794_DI_Flt ,
         SC_Local       := SL_22_P ,
         CM_ALM        := "dbPlcHmiALM".ALM[10257] ,
       );

NETWORK
TITLE = 10258 - LCP93_A291_FN3796 - Humidifier 6 Fan 1  - Motor Disconnect

       CALL #"LCP93_A291_FN3796"
       (
         CM_No       := 10258 ,
         Tab       := 22 ,
         SubTab       := 6 ,
         CfgType       := 0 ,
         CfgInvert       := True ,
         InputRaw       := LCP93_A291_FN3796_DI_Flt ,
         SC_Local       := SL_22_P ,
         CM_ALM        := "dbPlcHmiALM".ALM[10258] ,
       );

NETWORK
TITLE = 10259 - LCP93_A292_FN3797 - Humidifier 6 Fan 2  - Motor Disconnect

       CALL #"LCP93_A292_FN3797"
       (
         CM_No       := 10259 ,
         Tab       := 22 ,
         SubTab       := 6 ,
         CfgType       := 0 ,
         CfgInvert       := True ,
         InputRaw       := LCP93_A292_FN3797_DI_Flt ,
         SC_Local       := SL_22_P ,
         CM_ALM        := "dbPlcHmiALM".ALM[10259] ,
       );

NETWORK
TITLE = 10260 - LCP93_A293_FN3798 - Humidifier 6 Fan 3  - Motor Disconnect

       CALL #"LCP93_A293_FN3798"
       (
         CM_No       := 10260 ,
         Tab       := 22 ,
         SubTab       := 6 ,
         CfgType       := 0 ,
         CfgInvert       := True ,
         InputRaw       := LCP93_A293_FN3798_DI_Flt ,
         SC_Local       := SL_22_P ,
         CM_ALM        := "dbPlcHmiALM".ALM[10260] ,
       );

NETWORK
TITLE = 10261 - LCP93_A294_FN3799 - Humidifier 6 Fan 4 - Motor Disconnect

       CALL #"LCP93_A294_FN3799"
       (
         CM_No       := 10261 ,
         Tab       := 22 ,
         SubTab       := 6 ,
         CfgType       := 0 ,
         CfgInvert       := True ,
         InputRaw       := LCP93_A294_FN3799_DI_Flt ,
         SC_Local       := SL_22_P ,
         CM_ALM        := "dbPlcHmiALM".ALM[10261] ,
       );

NETWORK
TITLE = 10262 - LCP93_A170_BG7830 - Door 1 Humidifier 1 - Fan Room

       CALL #"LCP93_A170_BG7830"
       (
         CM_No       := 10262 ,
         Tab       := 1 ,
         SubTab       := 3 ,
         CfgType       := 0 ,
         CfgInvert       := True ,
         InputRaw       := LCP93_A170_BG7830_DI_ChA ,
         SC_Local       := SL_22_P ,
         CM_ALM        := "dbPlcHmiALM".ALM[10262] ,
       );

NETWORK
TITLE = 10263 - LCP93_A190_BG7832 - Door 1 Humidifier 3 - Fan Room

       CALL #"LCP93_A190_BG7832"
       (
         CM_No       := 10263 ,
         Tab       := 1 ,
         SubTab       := 3 ,
         CfgType       := 0 ,
         CfgInvert       := True ,
         InputRaw       := LCP93_A190_BG7832_DI_ChA ,
         SC_Local       := SL_22_P ,
         CM_ALM        := "dbPlcHmiALM".ALM[10263] ,
       );

NETWORK
TITLE = 10264 - LCP93_A270_BG7834 - Door 1 Humidifier 4 - Fan Room

       CALL #"LCP93_A270_BG7834"
       (
         CM_No       := 10264 ,
         Tab       := 1 ,
         SubTab       := 3 ,
         CfgType       := 0 ,
         CfgInvert       := True ,
         InputRaw       := LCP93_A270_BG7834_DI_ChA ,
         SC_Local       := SL_22_P ,
         CM_ALM        := "dbPlcHmiALM".ALM[10264] ,
       );

NETWORK
TITLE = 10265 - LCP93_A280_BG7836 - Door 1 Humidifier 5 - Fan Room

       CALL #"LCP93_A280_BG7836"
       (
         CM_No       := 10265 ,
         Tab       := 1 ,
         SubTab       := 3 ,
         CfgType       := 0 ,
         CfgInvert       := True ,
         InputRaw       := LCP93_A280_BG7836_DI_ChA ,
         SC_Local       := SL_22_P ,
         CM_ALM        := "dbPlcHmiALM".ALM[10265] ,
       );

NETWORK
TITLE = 10266 - LCP93_A290_BG7838 - Door 1 Humidifier 6 - Fan Room

       CALL #"LCP93_A290_BG7838"
       (
         CM_No       := 10266 ,
         Tab       := 1 ,
         SubTab       := 3 ,
         CfgType       := 0 ,
         CfgInvert       := True ,
         InputRaw       := LCP93_A290_BG7838_DI_ChA ,
         SC_Local       := SL_22_P ,
         CM_ALM        := "dbPlcHmiALM".ALM[10266] ,
       );

NETWORK
TITLE = 10267 - LCP93_ES01_SF6146 - Emergency Stop  - Humidifier Area

       CALL #"LCP93_ES01_SF6146"
       (
         CM_No       := 10267 ,
         Tab       := 1 ,
         SubTab       := 3 ,
         CfgType       := 0 ,
         CfgInvert       := True ,
         InputRaw       := LCP93_ES01_SF6146_DI_ChA ,
         SC_Local       := SL_01 ,
         CM_ALM        := "dbPlcHmiALM".ALM[10267] ,
       );

NETWORK
TITLE = 10268 - LCP93_ES01_SF6147 - Emergency Stop  - Humidifier Area

       CALL #"LCP93_ES01_SF6147"
       (
         CM_No       := 10268 ,
         Tab       := 1 ,
         SubTab       := 3 ,
         CfgType       := 0 ,
         CfgInvert       := True ,
         InputRaw       := LCP93_ES01_SF6147_DI_ChA ,
         SC_Local       := SL_01 ,
         CM_ALM        := "dbPlcHmiALM".ALM[10268] ,
       );

NETWORK
TITLE = 10269 - LCP93_ES01_SF6148 - Emergency Stop  - Humidifier Area

       CALL #"LCP93_ES01_SF6148"
       (
         CM_No       := 10269 ,
         Tab       := 1 ,
         SubTab       := 3 ,
         CfgType       := 0 ,
         CfgInvert       := True ,
         InputRaw       := LCP93_ES01_SF6148_DI_ChA ,
         SC_Local       := SL_01 ,
         CM_ALM        := "dbPlcHmiALM".ALM[10269] ,
       );

NETWORK
TITLE = 10270 - LCP93_ES01_SF6149 - Emergency Stop  - LCP93

       CALL #"LCP93_ES01_SF6149"
       (
         CM_No       := 10270 ,
         Tab       := 1 ,
         SubTab       := 3 ,
         CfgType       := 0 ,
         CfgInvert       := True ,
         InputRaw       := LCP93_ES01_SF6149_DI_ChA ,
         SC_Local       := SL_01 ,
         CM_ALM        := "dbPlcHmiALM".ALM[10270] ,
       );

NETWORK
TITLE = 10271 - LCP93_DC01_FC1000 - Power Feed Module 24VDC - Status

       CALL #"LCP93_DC01_FC1000"
       (
         CM_No       := 10271 ,
         Tab       := 13 ,
         SubTab       := 5 ,
         CfgType       := 0 ,
         CfgInvert       := True ,
         InputRaw       := LCP93_DC01_FC1000_DI_Flt ,
         SC_Local       := SL_13 ,
         CM_ALM        := "dbPlcHmiALM".ALM[10271] ,
       );

NETWORK
TITLE = 10272 - LCP93_IO_KF1000 - Point IO - EtherNet/IP Adapter

       CALL #"LCP93_IO_KF1000"
       (
         CM_No       := 10272 ,
         Tab       := 13 ,
         SubTab       := 5 ,
         CfgType       := 0 ,
         CfgInvert       := True ,
         InputRaw       :=  ,
         SC_Local       := SL_13 ,
         CM_ALM        := "dbPlcHmiALM".ALM[10272] ,
       );

NETWORK
TITLE = 10273 - LCP93_IO_KF3020 - 24V DC 8-Point Safety Input Module - SDI

       CALL #"LCP93_IO_KF3020"
       (
         CM_No       := 10273 ,
         Tab       := 13 ,
         SubTab       := 5 ,
         CfgType       := 0 ,
         CfgInvert       := True ,
         InputRaw       :=  ,
         SC_Local       := SL_13 ,
         CM_ALM        := "dbPlcHmiALM".ALM[10273] ,
       );

NETWORK
TITLE = 10274 - LCP93_IO_KF3021 - 24V DC 8-Point Safety Input Module - SDI

       CALL #"LCP93_IO_KF3021"
       (
         CM_No       := 10274 ,
         Tab       := 13 ,
         SubTab       := 5 ,
         CfgType       := 0 ,
         CfgInvert       := True ,
         InputRaw       :=  ,
         SC_Local       := SL_13 ,
         CM_ALM        := "dbPlcHmiALM".ALM[10274] ,
       );

NETWORK
TITLE = 10275 - LCP93_IO_KF3022 - 24V DC 8-Point Safety Input Module - SDI

       CALL #"LCP93_IO_KF3022"
       (
         CM_No       := 10275 ,
         Tab       := 13 ,
         SubTab       := 5 ,
         CfgType       := 0 ,
         CfgInvert       := True ,
         InputRaw       :=  ,
         SC_Local       := SL_13 ,
         CM_ALM        := "dbPlcHmiALM".ALM[10275] ,
       );

NETWORK
TITLE = 10276 - LCP101_AC01_FC3101 - 115VAC Power Supply - Thermal Fault

       CALL #"LCP101_AC01_FC3101"
       (
         CM_No       := 10276 ,
         Tab       := 13 ,
         SubTab       := 6 ,
         CfgType       := 0 ,
         CfgInvert       := True ,
         InputRaw       := LCP101_AC01_FC3101_DI_Flt ,
         SC_Local       := SL_13 ,
         CM_ALM        := "dbPlcHmiALM".ALM[10276] ,
       );

NETWORK
TITLE = 10277 - LCP101_I610_QA1101 - Min Gas Pressure Switch - (-BP8101)

       CALL #"LCP101_I610_QA1101"
       (
         CM_No       := 10277 ,
         Tab       := 28 ,
         SubTab       := 3 ,
         CfgType       := 0 ,
         CfgInvert       := True ,
         InputRaw       := LCP101_I610_QA1101_DI_FltL ,
         SC_Local       := SL_28_S1 ,
         CM_ALM        := "dbPlcHmiALM".ALM[10277] ,
       );

NETWORK
TITLE = 10278 - LCP101_I610_QA1102 - Max Gas Pressure Switch - (-BP8102)

       CALL #"LCP101_I610_QA1102"
       (
         CM_No       := 10278 ,
         Tab       := 28 ,
         SubTab       := 3 ,
         CfgType       := 0 ,
         CfgInvert       := True ,
         InputRaw       := LCP101_I610_QA1102_DI_FltH ,
         SC_Local       := SL_28_S1 ,
         CM_ALM        := "dbPlcHmiALM".ALM[10278] ,
       );

NETWORK
TITLE = 10279 - LCP101_I610_QA1103 - Leak Gas Pressure Switch - (-BP8103)

       CALL #"LCP101_I610_QA1103"
       (
         CM_No       := 10279 ,
         Tab       := 28 ,
         SubTab       := 3 ,
         CfgType       := 0 ,
         CfgInvert       := True ,
         InputRaw       := LCP101_I610_QA1103_DI_Ps ,
         SC_Local       := SL_28_S1 ,
         CM_ALM        := "dbPlcHmiALM".ALM[10279] ,
       );

NETWORK
TITLE = 10280 - LCP101_I610_QA1113 - No Air Check Pressure Switch - (-BP2113)

       CALL #"LCP101_I610_QA1113"
       (
         CM_No       := 10280 ,
         Tab       := 28 ,
         SubTab       := 3 ,
         CfgType       := 0 ,
         CfgInvert       := True ,
         InputRaw       := LCP101_I610_QA1113_DI_Ps ,
         SC_Local       := SL_28_S1 ,
         CM_ALM        := "dbPlcHmiALM".ALM[10280] ,
       );

NETWORK
TITLE = 10281 - LCP101_I610_QA1108 - Burner Failure - Signal from Maxon

       CALL #"LCP101_I610_QA1108"
       (
         CM_No       := 10281 ,
         Tab       := 28 ,
         SubTab       := 3 ,
         CfgType       := 0 ,
         CfgInvert       := True ,
         InputRaw       := LCP101_I610_QA1108_DI_Flt ,
         SC_Local       := SL_28_S1 ,
         CM_ALM        := "dbPlcHmiALM".ALM[10281] ,
       );

NETWORK
TITLE = 10282 - LCP101_I610_QA1104 - High Temperature Failure - Signal from JUMO

       CALL #"LCP101_I610_QA1104"
       (
         CM_No       := 10282 ,
         Tab       := 28 ,
         SubTab       := 3 ,
         CfgType       := 0 ,
         CfgInvert       := True ,
         InputRaw       := LCP101_I610_QA1104_DI_Flt ,
         SC_Local       := SL_28_S1 ,
         CM_ALM        := "dbPlcHmiALM".ALM[10282] ,
       );

NETWORK
TITLE = 10283 - LCP101_I512_BG7101 - Disc Filter 1 Door 1 - Before Filter

       CALL #"LCP101_I512_BG7101"
       (
         CM_No       := 10283 ,
         Tab       := 1 ,
         SubTab       := 8 ,
         CfgType       := 0 ,
         CfgInvert       := True ,
         InputRaw       := LCP101_I512_BG7101_DI_ChA ,
         SC_Local       := SL_28_S1 ,
         CM_ALM        := "dbPlcHmiALM".ALM[10283] ,
       );

NETWORK
TITLE = 10284 - LCP101_I512_BG7103 - Disc Filter 1 Door 2 - After Filter

       CALL #"LCP101_I512_BG7103"
       (
         CM_No       := 10284 ,
         Tab       := 1 ,
         SubTab       := 8 ,
         CfgType       := 0 ,
         CfgInvert       := True ,
         InputRaw       := LCP101_I512_BG7103_DI_ChA ,
         SC_Local       := SL_28_S1 ,
         CM_ALM        := "dbPlcHmiALM".ALM[10284] ,
       );

NETWORK
TITLE = 10285 - LCP101_I611_BP1120 - Zone 1 Circulation Fan - Diff. Pressure Circ. Fan 1

       CALL #"LCP101_I611_BP1120"
       (
         CM_No       := 10285 ,
         Tab       := 28 ,
         SubTab       := 3 ,
         CfgType       := 0 ,
         CfgInvert       := True ,
         InputRaw       := LCP101_I611_BP1120_DI_Ps ,
         SC_Local       := SL_28_S1 ,
         CM_ALM        := "dbPlcHmiALM".ALM[10285] ,
       );

NETWORK
TITLE = 10286 - LCP101_ES01_SF6151 - Emergency Stop  - Dryer 1 Zone 1 Area

       CALL #"LCP101_ES01_SF6151"
       (
         CM_No       := 10286 ,
         Tab       := 1 ,
         SubTab       := 5 ,
         CfgType       := 0 ,
         CfgInvert       := True ,
         InputRaw       := LCP101_ES01_SF6151_DI_ChA ,
         SC_Local       := SL_01 ,
         CM_ALM        := "dbPlcHmiALM".ALM[10286] ,
       );

NETWORK
TITLE = 10287 - LCP101_ES01_SF6152 - Emergency Stop  - LCP101

       CALL #"LCP101_ES01_SF6152"
       (
         CM_No       := 10287 ,
         Tab       := 1 ,
         SubTab       := 5 ,
         CfgType       := 0 ,
         CfgInvert       := True ,
         InputRaw       := LCP101_ES01_SF6152_DI_ChA ,
         SC_Local       := SL_01 ,
         CM_ALM        := "dbPlcHmiALM".ALM[10287] ,
       );

NETWORK
TITLE = 10288 - LCP101_DC01_FC1000 - Power Feed Module 24VDC - Status

       CALL #"LCP101_DC01_FC1000"
       (
         CM_No       := 10288 ,
         Tab       := 13 ,
         SubTab       := 6 ,
         CfgType       := 0 ,
         CfgInvert       := True ,
         InputRaw       := LCP101_DC01_FC1000_DI_Flt ,
         SC_Local       := SL_13 ,
         CM_ALM        := "dbPlcHmiALM".ALM[10288] ,
       );

NETWORK
TITLE = 10289 - LCP101_IO_KF1000 - Point IO - EtherNet/IP Adapter

       CALL #"LCP101_IO_KF1000"
       (
         CM_No       := 10289 ,
         Tab       := 13 ,
         SubTab       := 6 ,
         CfgType       := 0 ,
         CfgInvert       := True ,
         InputRaw       :=  ,
         SC_Local       := SL_13 ,
         CM_ALM        := "dbPlcHmiALM".ALM[10289] ,
       );

NETWORK
TITLE = 10290 - LCP101_IO_KF3013 - 24V DC 8-Point Safety Input Module - SDI

       CALL #"LCP101_IO_KF3013"
       (
         CM_No       := 10290 ,
         Tab       := 13 ,
         SubTab       := 6 ,
         CfgType       := 0 ,
         CfgInvert       := True ,
         InputRaw       :=  ,
         SC_Local       := SL_13 ,
         CM_ALM        := "dbPlcHmiALM".ALM[10290] ,
       );

NETWORK
TITLE = 10291 - LCP101_IO_KF3014 - 24V DC 8-Point Safety Input Module - SDI

       CALL #"LCP101_IO_KF3014"
       (
         CM_No       := 10291 ,
         Tab       := 13 ,
         SubTab       := 6 ,
         CfgType       := 0 ,
         CfgInvert       := True ,
         InputRaw       :=  ,
         SC_Local       := SL_13 ,
         CM_ALM        := "dbPlcHmiALM".ALM[10291] ,
       );

NETWORK
TITLE = 10292 - LCP102_AC01_FC3201 - 115VAC Power Supply - Thermal Fault

       CALL #"LCP102_AC01_FC3201"
       (
         CM_No       := 10292 ,
         Tab       := 13 ,
         SubTab       := 6 ,
         CfgType       := 0 ,
         CfgInvert       := True ,
         InputRaw       := LCP102_AC01_FC3201_DI_Flt ,
         SC_Local       := SL_13 ,
         CM_ALM        := "dbPlcHmiALM".ALM[10292] ,
       );

NETWORK
TITLE = 10293 - LCP102_I522_BG7201 - Disc Filter 2 Door 1 - Before Filter

       CALL #"LCP102_I522_BG7201"
       (
         CM_No       := 10293 ,
         Tab       := 1 ,
         SubTab       := 8 ,
         CfgType       := 0 ,
         CfgInvert       := True ,
         InputRaw       := LCP102_I522_BG7201_DI_ChA ,
         SC_Local       := SL_28_S1 ,
         CM_ALM        := "dbPlcHmiALM".ALM[10293] ,
       );

NETWORK
TITLE = 10294 - LCP102_I522_BG7203 - Disc Filter 2 Door 1 - After Filter

       CALL #"LCP102_I522_BG7203"
       (
         CM_No       := 10294 ,
         Tab       := 1 ,
         SubTab       := 8 ,
         CfgType       := 0 ,
         CfgInvert       := True ,
         InputRaw       := LCP102_I522_BG7203_DI_ChA ,
         SC_Local       := SL_28_S1 ,
         CM_ALM        := "dbPlcHmiALM".ALM[10294] ,
       );

NETWORK
TITLE = 10295 - LCP102_I621_BP1222 - Zone 2 Circulation Fan - Diff. Pressure Circ. Fan 2

       CALL #"LCP102_I621_BP1222"
       (
         CM_No       := 10295 ,
         Tab       := 28 ,
         SubTab       := 4 ,
         CfgType       := 0 ,
         CfgInvert       := True ,
         InputRaw       := LCP102_I621_BP1222_DI_Ps ,
         SC_Local       := SL_28_S1 ,
         CM_ALM        := "dbPlcHmiALM".ALM[10295] ,
       );

NETWORK
TITLE = 10296 - LCP102_ES01_SF6253 - Emergency Stop  - Dryer 1 Zone 2 Area

       CALL #"LCP102_ES01_SF6253"
       (
         CM_No       := 10296 ,
         Tab       := 1 ,
         SubTab       := 5 ,
         CfgType       := 0 ,
         CfgInvert       := True ,
         InputRaw       := LCP102_ES01_SF6253_DI_ChA ,
         SC_Local       := SL_01 ,
         CM_ALM        := "dbPlcHmiALM".ALM[10296] ,
       );

NETWORK
TITLE = 10297 - LCP102_ES01_SF6254 - Emergency Stop  - LCP102

       CALL #"LCP102_ES01_SF6254"
       (
         CM_No       := 10297 ,
         Tab       := 1 ,
         SubTab       := 5 ,
         CfgType       := 0 ,
         CfgInvert       := True ,
         InputRaw       := LCP102_ES01_SF6254_DI_ChA ,
         SC_Local       := SL_01 ,
         CM_ALM        := "dbPlcHmiALM".ALM[10297] ,
       );

NETWORK
TITLE = 10298 - LCP102_DC01_FC1000 - Power Feed Module 24VDC - Status

       CALL #"LCP102_DC01_FC1000"
       (
         CM_No       := 10298 ,
         Tab       := 13 ,
         SubTab       := 6 ,
         CfgType       := 0 ,
         CfgInvert       := True ,
         InputRaw       := LCP102_DC01_FC1000_DI_Flt ,
         SC_Local       := SL_13 ,
         CM_ALM        := "dbPlcHmiALM".ALM[10298] ,
       );

NETWORK
TITLE = 10299 - LCP102_IO_KF1000 - Point IO - EtherNet/IP Adapter

       CALL #"LCP102_IO_KF1000"
       (
         CM_No       := 10299 ,
         Tab       := 13 ,
         SubTab       := 6 ,
         CfgType       := 0 ,
         CfgInvert       := True ,
         InputRaw       :=  ,
         SC_Local       := SL_13 ,
         CM_ALM        := "dbPlcHmiALM".ALM[10299] ,
       );

NETWORK
TITLE = 10300 - LCP102_IO_KF3008 - 24V DC 8-Point Safety Input Module - SDI

       CALL #"LCP102_IO_KF3008"
       (
         CM_No       := 10300 ,
         Tab       := 13 ,
         SubTab       := 6 ,
         CfgType       := 0 ,
         CfgInvert       := True ,
         InputRaw       :=  ,
         SC_Local       := SL_13 ,
         CM_ALM        := "dbPlcHmiALM".ALM[10300] ,
       );

NETWORK
TITLE = 10301 - LCP102_IO_KF3009 - 24V DC 8-Point Safety Input Module - SDI

       CALL #"LCP102_IO_KF3009"
       (
         CM_No       := 10301 ,
         Tab       := 13 ,
         SubTab       := 6 ,
         CfgType       := 0 ,
         CfgInvert       := True ,
         InputRaw       :=  ,
         SC_Local       := SL_13 ,
         CM_ALM        := "dbPlcHmiALM".ALM[10301] ,
       );

NETWORK
TITLE = 10302 - LCP102_IO_KF3010 - 24V DC 8-Point Source Safety Output Module - SDO

       CALL #"LCP102_IO_KF3010"
       (
         CM_No       := 10302 ,
         Tab       := 13 ,
         SubTab       := 6 ,
         CfgType       := 0 ,
         CfgInvert       := True ,
         InputRaw       :=  ,
         SC_Local       := SL_13 ,
         CM_ALM        := "dbPlcHmiALM".ALM[10302] ,
       );

NETWORK
TITLE = 10303 - LCP103_AC01_FC3301 - 115VAC Power Supply - Thermal Fault

       CALL #"LCP103_AC01_FC3301"
       (
         CM_No       := 10303 ,
         Tab       := 13 ,
         SubTab       := 6 ,
         CfgType       := 0 ,
         CfgInvert       := True ,
         InputRaw       := LCP103_AC01_FC3301_DI_Flt ,
         SC_Local       := SL_13 ,
         CM_ALM        := "dbPlcHmiALM".ALM[10303] ,
       );

NETWORK
TITLE = 10304 - LCP103_I630_QA1301 - Min Gas Pressure Switch - (-BP8301)

       CALL #"LCP103_I630_QA1301"
       (
         CM_No       := 10304 ,
         Tab       := 28 ,
         SubTab       := 5 ,
         CfgType       := 0 ,
         CfgInvert       := True ,
         InputRaw       := LCP103_I630_QA1301_DI_FltL ,
         SC_Local       := SL_28_S2 ,
         CM_ALM        := "dbPlcHmiALM".ALM[10304] ,
       );

NETWORK
TITLE = 10305 - LCP103_I630_QA1302 - Max Gas Pressure Switch - (-BP8302)

       CALL #"LCP103_I630_QA1302"
       (
         CM_No       := 10305 ,
         Tab       := 28 ,
         SubTab       := 5 ,
         CfgType       := 0 ,
         CfgInvert       := True ,
         InputRaw       := LCP103_I630_QA1302_DI_FltH ,
         SC_Local       := SL_28_S2 ,
         CM_ALM        := "dbPlcHmiALM".ALM[10305] ,
       );

NETWORK
TITLE = 10306 - LCP103_I630_QA1303 - Leak Gas Pressure Switch - (-BP8303)

       CALL #"LCP103_I630_QA1303"
       (
         CM_No       := 10306 ,
         Tab       := 28 ,
         SubTab       := 5 ,
         CfgType       := 0 ,
         CfgInvert       := True ,
         InputRaw       := LCP103_I630_QA1303_DI_Ps ,
         SC_Local       := SL_28_S2 ,
         CM_ALM        := "dbPlcHmiALM".ALM[10306] ,
       );

NETWORK
TITLE = 10307 - LCP103_I630_QA1313 - No Air Check Pressure Switch - (-BP2313)

       CALL #"LCP103_I630_QA1313"
       (
         CM_No       := 10307 ,
         Tab       := 28 ,
         SubTab       := 5 ,
         CfgType       := 0 ,
         CfgInvert       := True ,
         InputRaw       := LCP103_I630_QA1313_DI_Ps ,
         SC_Local       := SL_28_S2 ,
         CM_ALM        := "dbPlcHmiALM".ALM[10307] ,
       );

NETWORK
TITLE = 10308 - LCP103_I630_QA1308 - Burner Failure - Signal from Maxon

       CALL #"LCP103_I630_QA1308"
       (
         CM_No       := 10308 ,
         Tab       := 28 ,
         SubTab       := 5 ,
         CfgType       := 0 ,
         CfgInvert       := True ,
         InputRaw       := LCP103_I630_QA1308_DI_Flt ,
         SC_Local       := SL_28_S2 ,
         CM_ALM        := "dbPlcHmiALM".ALM[10308] ,
       );

NETWORK
TITLE = 10309 - LCP103_I630_QA1304 - High Temperature Failure - Signal from JUMO

       CALL #"LCP103_I630_QA1304"
       (
         CM_No       := 10309 ,
         Tab       := 28 ,
         SubTab       := 5 ,
         CfgType       := 0 ,
         CfgInvert       := True ,
         InputRaw       := LCP103_I630_QA1304_DI_Flt ,
         SC_Local       := SL_28_S2 ,
         CM_ALM        := "dbPlcHmiALM".ALM[10309] ,
       );

NETWORK
TITLE = 10310 - LCP103_K512_BG7301 - Disc Filter 3 Door 1 - Before Filter

       CALL #"LCP103_K512_BG7301"
       (
         CM_No       := 10310 ,
         Tab       := 1 ,
         SubTab       := 8 ,
         CfgType       := 0 ,
         CfgInvert       := True ,
         InputRaw       := LCP103_K512_BG7301_DI_ChA ,
         SC_Local       := SL_28_S2 ,
         CM_ALM        := "dbPlcHmiALM".ALM[10310] ,
       );

NETWORK
TITLE = 10311 - LCP103_K512_BG7303 - Disc Filter 3 Door 2 - After Filter

       CALL #"LCP103_K512_BG7303"
       (
         CM_No       := 10311 ,
         Tab       := 1 ,
         SubTab       := 8 ,
         CfgType       := 0 ,
         CfgInvert       := True ,
         InputRaw       := LCP103_K512_BG7303_DI_ChA ,
         SC_Local       := SL_28_S2 ,
         CM_ALM        := "dbPlcHmiALM".ALM[10311] ,
       );

NETWORK
TITLE = 10312 - LCP103_K611_BP1323 - Zone 3 Circulation Fan - Diff. Pressure Circ. Fan 3

       CALL #"LCP103_K611_BP1323"
       (
         CM_No       := 10312 ,
         Tab       := 28 ,
         SubTab       := 5 ,
         CfgType       := 0 ,
         CfgInvert       := True ,
         InputRaw       := LCP103_K611_BP1323_DI_Ps ,
         SC_Local       := SL_28_S2 ,
         CM_ALM        := "dbPlcHmiALM".ALM[10312] ,
       );

NETWORK
TITLE = 10313 - LCP103_ES01_SF6355 - Emergency Stop  - Dryer 2 Zone 3 Area

       CALL #"LCP103_ES01_SF6355"
       (
         CM_No       := 10313 ,
         Tab       := 1 ,
         SubTab       := 5 ,
         CfgType       := 0 ,
         CfgInvert       := True ,
         InputRaw       := LCP103_ES01_SF6355_DI_ChA ,
         SC_Local       := SL_01 ,
         CM_ALM        := "dbPlcHmiALM".ALM[10313] ,
       );

NETWORK
TITLE = 10314 - LCP103_ES01_SF6356 - Emergency Stop  - LCP103

       CALL #"LCP103_ES01_SF6356"
       (
         CM_No       := 10314 ,
         Tab       := 1 ,
         SubTab       := 5 ,
         CfgType       := 0 ,
         CfgInvert       := True ,
         InputRaw       := LCP103_ES01_SF6356_DI_ChA ,
         SC_Local       := SL_01 ,
         CM_ALM        := "dbPlcHmiALM".ALM[10314] ,
       );

NETWORK
TITLE = 10315 - LCP103_DC01_FC1000 - Power Feed Module 24VDC - Status

       CALL #"LCP103_DC01_FC1000"
       (
         CM_No       := 10315 ,
         Tab       := 13 ,
         SubTab       := 6 ,
         CfgType       := 0 ,
         CfgInvert       := True ,
         InputRaw       := LCP103_DC01_FC1000_DI_Flt ,
         SC_Local       := SL_13 ,
         CM_ALM        := "dbPlcHmiALM".ALM[10315] ,
       );

NETWORK
TITLE = 10316 - LCP103_IO_KF1000 - Point IO - EtherNet/IP Adapter

       CALL #"LCP103_IO_KF1000"
       (
         CM_No       := 10316 ,
         Tab       := 13 ,
         SubTab       := 6 ,
         CfgType       := 0 ,
         CfgInvert       := True ,
         InputRaw       :=  ,
         SC_Local       := SL_13 ,
         CM_ALM        := "dbPlcHmiALM".ALM[10316] ,
       );

NETWORK
TITLE = 10317 - LCP103_IO_KF3013 - 24V DC 8-Point Safety Input Module - SDI

       CALL #"LCP103_IO_KF3013"
       (
         CM_No       := 10317 ,
         Tab       := 13 ,
         SubTab       := 6 ,
         CfgType       := 0 ,
         CfgInvert       := True ,
         InputRaw       :=  ,
         SC_Local       := SL_13 ,
         CM_ALM        := "dbPlcHmiALM".ALM[10317] ,
       );

NETWORK
TITLE = 10318 - LCP103_IO_KF3014 - 24V DC 8-Point Safety Input Module - SDI

       CALL #"LCP103_IO_KF3014"
       (
         CM_No       := 10318 ,
         Tab       := 13 ,
         SubTab       := 6 ,
         CfgType       := 0 ,
         CfgInvert       := True ,
         InputRaw       :=  ,
         SC_Local       := SL_13 ,
         CM_ALM        := "dbPlcHmiALM".ALM[10318] ,
       );

NETWORK
TITLE = 10319 - LCP104_AC01_FC3401 - 115VAC Power Supply - Thermal Fault

       CALL #"LCP104_AC01_FC3401"
       (
         CM_No       := 10319 ,
         Tab       := 13 ,
         SubTab       := 6 ,
         CfgType       := 0 ,
         CfgInvert       := True ,
         InputRaw       := LCP104_AC01_FC3401_DI_Flt ,
         SC_Local       := SL_13 ,
         CM_ALM        := "dbPlcHmiALM".ALM[10319] ,
       );

NETWORK
TITLE = 10320 - LCP104_I640_QA1401 - Min Gas Pressure Switch - (-BP8401)

       CALL #"LCP104_I640_QA1401"
       (
         CM_No       := 10320 ,
         Tab       := 28 ,
         SubTab       := 6 ,
         CfgType       := 0 ,
         CfgInvert       := True ,
         InputRaw       := LCP104_I640_QA1401_DI_FltL ,
         SC_Local       := SL_28_S2 ,
         CM_ALM        := "dbPlcHmiALM".ALM[10320] ,
       );

NETWORK
TITLE = 10321 - LCP104_I640_QA1402 - Max Gas Pressure Switch - (-BP8402)

       CALL #"LCP104_I640_QA1402"
       (
         CM_No       := 10321 ,
         Tab       := 28 ,
         SubTab       := 6 ,
         CfgType       := 0 ,
         CfgInvert       := True ,
         InputRaw       := LCP104_I640_QA1402_DI_FltH ,
         SC_Local       := SL_28_S2 ,
         CM_ALM        := "dbPlcHmiALM".ALM[10321] ,
       );

NETWORK
TITLE = 10322 - LCP104_I640_QA1403 - Leak Gas Pressure Switch - (-BP8403)

       CALL #"LCP104_I640_QA1403"
       (
         CM_No       := 10322 ,
         Tab       := 28 ,
         SubTab       := 6 ,
         CfgType       := 0 ,
         CfgInvert       := True ,
         InputRaw       := LCP104_I640_QA1403_DI_Ps ,
         SC_Local       := SL_28_S2 ,
         CM_ALM        := "dbPlcHmiALM".ALM[10322] ,
       );

NETWORK
TITLE = 10323 - LCP104_I640_QA1413 - No Air Check Pressure Switch - (-BP2413)

       CALL #"LCP104_I640_QA1413"
       (
         CM_No       := 10323 ,
         Tab       := 28 ,
         SubTab       := 6 ,
         CfgType       := 0 ,
         CfgInvert       := True ,
         InputRaw       := LCP104_I640_QA1413_DI_Ps ,
         SC_Local       := SL_28_S2 ,
         CM_ALM        := "dbPlcHmiALM".ALM[10323] ,
       );

NETWORK
TITLE = 10324 - LCP104_I640_QA1408 - Burner Failure - Signal from Maxon

       CALL #"LCP104_I640_QA1408"
       (
         CM_No       := 10324 ,
         Tab       := 28 ,
         SubTab       := 6 ,
         CfgType       := 0 ,
         CfgInvert       := True ,
         InputRaw       := LCP104_I640_QA1408_DI_Flt ,
         SC_Local       := SL_28_S2 ,
         CM_ALM        := "dbPlcHmiALM".ALM[10324] ,
       );

NETWORK
TITLE = 10325 - LCP104_I640_QA1404 - High Temperature Failure - Signal from JUMO

       CALL #"LCP104_I640_QA1404"
       (
         CM_No       := 10325 ,
         Tab       := 28 ,
         SubTab       := 6 ,
         CfgType       := 0 ,
         CfgInvert       := True ,
         InputRaw       := LCP104_I640_QA1404_DI_Flt ,
         SC_Local       := SL_28_S2 ,
         CM_ALM        := "dbPlcHmiALM".ALM[10325] ,
       );

NETWORK
TITLE = 10326 - LCP104_K522_BG7401 - Disc Filter 4 Door 1 - Before Filter

       CALL #"LCP104_K522_BG7401"
       (
         CM_No       := 10326 ,
         Tab       := 1 ,
         SubTab       := 8 ,
         CfgType       := 0 ,
         CfgInvert       := True ,
         InputRaw       := LCP104_K522_BG7401_DI_ChA ,
         SC_Local       := SL_28_S2 ,
         CM_ALM        := "dbPlcHmiALM".ALM[10326] ,
       );

NETWORK
TITLE = 10327 - LCP104_K522_BG7403 - Disc Filter 4 Door 2 - After Filter

       CALL #"LCP104_K522_BG7403"
       (
         CM_No       := 10327 ,
         Tab       := 1 ,
         SubTab       := 8 ,
         CfgType       := 0 ,
         CfgInvert       := True ,
         InputRaw       := LCP104_K522_BG7403_DI_ChA ,
         SC_Local       := SL_28_S2 ,
         CM_ALM        := "dbPlcHmiALM".ALM[10327] ,
       );

NETWORK
TITLE = 10328 - LCP104_K621_BP1424 - Zone 4 Circulation Fan  - Diff. Pressure Circ. Fan 4

       CALL #"LCP104_K621_BP1424"
       (
         CM_No       := 10328 ,
         Tab       := 28 ,
         SubTab       := 6 ,
         CfgType       := 0 ,
         CfgInvert       := True ,
         InputRaw       := LCP104_K621_BP1424_DI_Ps ,
         SC_Local       := SL_28_S2 ,
         CM_ALM        := "dbPlcHmiALM".ALM[10328] ,
       );

NETWORK
TITLE = 10329 - LCP104_ES01_SF6457 - Emergency Stop  - Dryer 2 Zone 4 Area

       CALL #"LCP104_ES01_SF6457"
       (
         CM_No       := 10329 ,
         Tab       := 1 ,
         SubTab       := 5 ,
         CfgType       := 0 ,
         CfgInvert       := True ,
         InputRaw       := LCP104_ES01_SF6457_DI_ChA ,
         SC_Local       := SL_01 ,
         CM_ALM        := "dbPlcHmiALM".ALM[10329] ,
       );

NETWORK
TITLE = 10330 - LCP104_ES01_SF6458 - Emergency Stop  - LCP104

       CALL #"LCP104_ES01_SF6458"
       (
         CM_No       := 10330 ,
         Tab       := 1 ,
         SubTab       := 5 ,
         CfgType       := 0 ,
         CfgInvert       := True ,
         InputRaw       := LCP104_ES01_SF6458_DI_ChA ,
         SC_Local       := SL_01 ,
         CM_ALM        := "dbPlcHmiALM".ALM[10330] ,
       );

NETWORK
TITLE = 10331 - LCP104_DC01_FC1000 - Power Feed Module 24VDC - Status

       CALL #"LCP104_DC01_FC1000"
       (
         CM_No       := 10331 ,
         Tab       := 13 ,
         SubTab       := 6 ,
         CfgType       := 0 ,
         CfgInvert       := True ,
         InputRaw       := LCP104_DC01_FC1000_DI_Flt ,
         SC_Local       := SL_13 ,
         CM_ALM        := "dbPlcHmiALM".ALM[10331] ,
       );

NETWORK
TITLE = 10332 - LCP104_IO_KF1000 - Point IO - EtherNet/IP Adapter

       CALL #"LCP104_IO_KF1000"
       (
         CM_No       := 10332 ,
         Tab       := 13 ,
         SubTab       := 6 ,
         CfgType       := 0 ,
         CfgInvert       := True ,
         InputRaw       :=  ,
         SC_Local       := SL_13 ,
         CM_ALM        := "dbPlcHmiALM".ALM[10332] ,
       );

NETWORK
TITLE = 10333 - LCP104_IO_KF3013 - 24V DC 8-Point Safety Input Module - SDI

       CALL #"LCP104_IO_KF3013"
       (
         CM_No       := 10333 ,
         Tab       := 13 ,
         SubTab       := 6 ,
         CfgType       := 0 ,
         CfgInvert       := True ,
         InputRaw       :=  ,
         SC_Local       := SL_13 ,
         CM_ALM        := "dbPlcHmiALM".ALM[10333] ,
       );

NETWORK
TITLE = 10334 - LCP104_IO_KF3014 - 24V DC 8-Point Safety Input Module - SDI

       CALL #"LCP104_IO_KF3014"
       (
         CM_No       := 10334 ,
         Tab       := 13 ,
         SubTab       := 6 ,
         CfgType       := 0 ,
         CfgInvert       := True ,
         InputRaw       :=  ,
         SC_Local       := SL_13 ,
         CM_ALM        := "dbPlcHmiALM".ALM[10334] ,
       );

NETWORK
TITLE = 10335 - LCP111_AC01_FC3501 - 115VAC Power Supply - Thermal Fault

       CALL #"LCP111_AC01_FC3501"
       (
         CM_No       := 10335 ,
         Tab       := 13 ,
         SubTab       := 6 ,
         CfgType       := 0 ,
         CfgInvert       := True ,
         InputRaw       := LCP111_AC01_FC3501_DI_Flt ,
         SC_Local       := SL_13 ,
         CM_ALM        := "dbPlcHmiALM".ALM[10335] ,
       );

NETWORK
TITLE = 10336 - LCP111_I650_QA1501 - Min Gas Pressure Switch - (-BP8501)

       CALL #"LCP111_I650_QA1501"
       (
         CM_No       := 10336 ,
         Tab       := 28 ,
         SubTab       := 7 ,
         CfgType       := 0 ,
         CfgInvert       := True ,
         InputRaw       := LCP111_I650_QA1501_DI_FltL ,
         SC_Local       := SL_28_S3 ,
         CM_ALM        := "dbPlcHmiALM".ALM[10336] ,
       );

NETWORK
TITLE = 10337 - LCP111_I650_QA1502 - Max Gas Pressure Switch - (-BP8502)

       CALL #"LCP111_I650_QA1502"
       (
         CM_No       := 10337 ,
         Tab       := 28 ,
         SubTab       := 7 ,
         CfgType       := 0 ,
         CfgInvert       := True ,
         InputRaw       := LCP111_I650_QA1502_DI_FltH ,
         SC_Local       := SL_28_S3 ,
         CM_ALM        := "dbPlcHmiALM".ALM[10337] ,
       );

NETWORK
TITLE = 10338 - LCP111_I650_QA1503 - Leak Gas Pressure Switch - (-BP8503)

       CALL #"LCP111_I650_QA1503"
       (
         CM_No       := 10338 ,
         Tab       := 28 ,
         SubTab       := 7 ,
         CfgType       := 0 ,
         CfgInvert       := True ,
         InputRaw       := LCP111_I650_QA1503_DI_Ps ,
         SC_Local       := SL_28_S3 ,
         CM_ALM        := "dbPlcHmiALM".ALM[10338] ,
       );

NETWORK
TITLE = 10339 - LCP111_I650_QA1513 - No Air Check Pressure Switch - (-BP2513)

       CALL #"LCP111_I650_QA1513"
       (
         CM_No       := 10339 ,
         Tab       := 28 ,
         SubTab       := 7 ,
         CfgType       := 0 ,
         CfgInvert       := True ,
         InputRaw       := LCP111_I650_QA1513_DI_Ps ,
         SC_Local       := SL_28_S3 ,
         CM_ALM        := "dbPlcHmiALM".ALM[10339] ,
       );

NETWORK
TITLE = 10340 - LCP111_I650_QA1508 - Burner Failure - Signal from Maxon

       CALL #"LCP111_I650_QA1508"
       (
         CM_No       := 10340 ,
         Tab       := 28 ,
         SubTab       := 7 ,
         CfgType       := 0 ,
         CfgInvert       := True ,
         InputRaw       := LCP111_I650_QA1508_DI_Flt ,
         SC_Local       := SL_28_S3 ,
         CM_ALM        := "dbPlcHmiALM".ALM[10340] ,
       );

NETWORK
TITLE = 10341 - LCP111_I650_QA1504 - High Temperature Failure - Signal from JUMO

       CALL #"LCP111_I650_QA1504"
       (
         CM_No       := 10341 ,
         Tab       := 28 ,
         SubTab       := 7 ,
         CfgType       := 0 ,
         CfgInvert       := True ,
         InputRaw       := LCP111_I650_QA1504_DI_Flt ,
         SC_Local       := SL_28_S3 ,
         CM_ALM        := "dbPlcHmiALM".ALM[10341] ,
       );

NETWORK
TITLE = 10342 - LCP111_N512_BG7501 - Disc Filter 5 Door 1 - Before Filter

       CALL #"LCP111_N512_BG7501"
       (
         CM_No       := 10342 ,
         Tab       := 1 ,
         SubTab       := 8 ,
         CfgType       := 0 ,
         CfgInvert       := True ,
         InputRaw       := LCP111_N512_BG7501_DI_ChA ,
         SC_Local       := SL_28_S3 ,
         CM_ALM        := "dbPlcHmiALM".ALM[10342] ,
       );

NETWORK
TITLE = 10343 - LCP111_N512_BG7503 - Disc Filter 5 Door 2 - After Filter

       CALL #"LCP111_N512_BG7503"
       (
         CM_No       := 10343 ,
         Tab       := 1 ,
         SubTab       := 8 ,
         CfgType       := 0 ,
         CfgInvert       := True ,
         InputRaw       := LCP111_N512_BG7503_DI_ChA ,
         SC_Local       := SL_28_S3 ,
         CM_ALM        := "dbPlcHmiALM".ALM[10343] ,
       );

NETWORK
TITLE = 10344 - LCP111_N611_BP1525 - Zone 5 Circulation Fan  - Diff. Pressure Circ. Fan 5

       CALL #"LCP111_N611_BP1525"
       (
         CM_No       := 10344 ,
         Tab       := 28 ,
         SubTab       := 7 ,
         CfgType       := 0 ,
         CfgInvert       := True ,
         InputRaw       := LCP111_N611_BP1525_DI_Ps ,
         SC_Local       := SL_28_S3 ,
         CM_ALM        := "dbPlcHmiALM".ALM[10344] ,
       );

NETWORK
TITLE = 10345 - LCP111_ES01_SF6559 - Emergency Stop  - Dryer 3 Zone 5 Area

       CALL #"LCP111_ES01_SF6559"
       (
         CM_No       := 10345 ,
         Tab       := 1 ,
         SubTab       := 6 ,
         CfgType       := 0 ,
         CfgInvert       := True ,
         InputRaw       := LCP111_ES01_SF6559_DI_ChA ,
         SC_Local       := SL_01 ,
         CM_ALM        := "dbPlcHmiALM".ALM[10345] ,
       );

NETWORK
TITLE = 10346 - LCP111_ES01_SF6560 - Emergency Stop  - LCP111

       CALL #"LCP111_ES01_SF6560"
       (
         CM_No       := 10346 ,
         Tab       := 1 ,
         SubTab       := 6 ,
         CfgType       := 0 ,
         CfgInvert       := True ,
         InputRaw       := LCP111_ES01_SF6560_DI_ChA ,
         SC_Local       := SL_01 ,
         CM_ALM        := "dbPlcHmiALM".ALM[10346] ,
       );

NETWORK
TITLE = 10347 - LCP111_DC01_FC1000 - Power Feed Module 24VDC - Status

       CALL #"LCP111_DC01_FC1000"
       (
         CM_No       := 10347 ,
         Tab       := 13 ,
         SubTab       := 6 ,
         CfgType       := 0 ,
         CfgInvert       := True ,
         InputRaw       := LCP111_DC01_FC1000_DI_Flt ,
         SC_Local       := SL_13 ,
         CM_ALM        := "dbPlcHmiALM".ALM[10347] ,
       );

NETWORK
TITLE = 10348 - LCP111_IO_KF1000 - Point IO - EtherNet/IP Adapter

       CALL #"LCP111_IO_KF1000"
       (
         CM_No       := 10348 ,
         Tab       := 13 ,
         SubTab       := 6 ,
         CfgType       := 0 ,
         CfgInvert       := True ,
         InputRaw       :=  ,
         SC_Local       := SL_13 ,
         CM_ALM        := "dbPlcHmiALM".ALM[10348] ,
       );

NETWORK
TITLE = 10349 - LCP111_IO_KF3013 - 24V DC 8-Point Safety Input Module - SDI

       CALL #"LCP111_IO_KF3013"
       (
         CM_No       := 10349 ,
         Tab       := 13 ,
         SubTab       := 6 ,
         CfgType       := 0 ,
         CfgInvert       := True ,
         InputRaw       :=  ,
         SC_Local       := SL_13 ,
         CM_ALM        := "dbPlcHmiALM".ALM[10349] ,
       );

NETWORK
TITLE = 10350 - LCP111_IO_KF3014 - 24V DC 8-Point Safety Input Module - SDI

       CALL #"LCP111_IO_KF3014"
       (
         CM_No       := 10350 ,
         Tab       := 13 ,
         SubTab       := 6 ,
         CfgType       := 0 ,
         CfgInvert       := True ,
         InputRaw       :=  ,
         SC_Local       := SL_13 ,
         CM_ALM        := "dbPlcHmiALM".ALM[10350] ,
       );

NETWORK
TITLE = 10351 - LCP112_AC01_FC3601 - 115VAC Power Supply - Thermal Fault

       CALL #"LCP112_AC01_FC3601"
       (
         CM_No       := 10351 ,
         Tab       := 13 ,
         SubTab       := 6 ,
         CfgType       := 0 ,
         CfgInvert       := True ,
         InputRaw       := LCP112_AC01_FC3601_DI_Flt ,
         SC_Local       := SL_13 ,
         CM_ALM        := "dbPlcHmiALM".ALM[10351] ,
       );

NETWORK
TITLE = 10352 - LCP112_I660_QA1601 - Min Gas Pressure Switch - (-BP8601)

       CALL #"LCP112_I660_QA1601"
       (
         CM_No       := 10352 ,
         Tab       := 28 ,
         SubTab       := 8 ,
         CfgType       := 0 ,
         CfgInvert       := True ,
         InputRaw       := LCP112_I660_QA1601_DI_FltL ,
         SC_Local       := SL_28_S3 ,
         CM_ALM        := "dbPlcHmiALM".ALM[10352] ,
       );

NETWORK
TITLE = 10353 - LCP112_I660_QA1602 - Max Gas Pressure Switch - (-BP8602)

       CALL #"LCP112_I660_QA1602"
       (
         CM_No       := 10353 ,
         Tab       := 28 ,
         SubTab       := 8 ,
         CfgType       := 0 ,
         CfgInvert       := True ,
         InputRaw       := LCP112_I660_QA1602_DI_FltH ,
         SC_Local       := SL_28_S3 ,
         CM_ALM        := "dbPlcHmiALM".ALM[10353] ,
       );

NETWORK
TITLE = 10354 - LCP112_I660_QA1603 - Leak Gas Pressure Switch - (-BP8603)

       CALL #"LCP112_I660_QA1603"
       (
         CM_No       := 10354 ,
         Tab       := 28 ,
         SubTab       := 8 ,
         CfgType       := 0 ,
         CfgInvert       := True ,
         InputRaw       := LCP112_I660_QA1603_DI_Ps ,
         SC_Local       := SL_28_S3 ,
         CM_ALM        := "dbPlcHmiALM".ALM[10354] ,
       );

NETWORK
TITLE = 10355 - LCP112_I660_QA1613 - No Air Check Pressure Switch - (-BP2613)

       CALL #"LCP112_I660_QA1613"
       (
         CM_No       := 10355 ,
         Tab       := 28 ,
         SubTab       := 8 ,
         CfgType       := 0 ,
         CfgInvert       := True ,
         InputRaw       := LCP112_I660_QA1613_DI_Ps ,
         SC_Local       := SL_28_S3 ,
         CM_ALM        := "dbPlcHmiALM".ALM[10355] ,
       );

NETWORK
TITLE = 10356 - LCP112_I660_QA1608 - Burner Failure - Signal from Maxon

       CALL #"LCP112_I660_QA1608"
       (
         CM_No       := 10356 ,
         Tab       := 28 ,
         SubTab       := 8 ,
         CfgType       := 0 ,
         CfgInvert       := True ,
         InputRaw       := LCP112_I660_QA1608_DI_Flt ,
         SC_Local       := SL_28_S3 ,
         CM_ALM        := "dbPlcHmiALM".ALM[10356] ,
       );

NETWORK
TITLE = 10357 - LCP112_I660_QA1604 - High Temperature Failure - Signal from JUMO

       CALL #"LCP112_I660_QA1604"
       (
         CM_No       := 10357 ,
         Tab       := 28 ,
         SubTab       := 8 ,
         CfgType       := 0 ,
         CfgInvert       := True ,
         InputRaw       := LCP112_I660_QA1604_DI_Flt ,
         SC_Local       := SL_28_S3 ,
         CM_ALM        := "dbPlcHmiALM".ALM[10357] ,
       );

NETWORK
TITLE = 10358 - LCP112_N522_BG7601 - Disc Filter 6 Door 1 - Before Filter

       CALL #"LCP112_N522_BG7601"
       (
         CM_No       := 10358 ,
         Tab       := 1 ,
         SubTab       := 8 ,
         CfgType       := 0 ,
         CfgInvert       := True ,
         InputRaw       := LCP112_N522_BG7601_DI_ChA ,
         SC_Local       := SL_28_S3 ,
         CM_ALM        := "dbPlcHmiALM".ALM[10358] ,
       );

NETWORK
TITLE = 10359 - LCP112_N522_BG7603 - Disc Filter 6 Door 2 - After Filter

       CALL #"LCP112_N522_BG7603"
       (
         CM_No       := 10359 ,
         Tab       := 1 ,
         SubTab       := 8 ,
         CfgType       := 0 ,
         CfgInvert       := True ,
         InputRaw       := LCP112_N522_BG7603_DI_ChA ,
         SC_Local       := SL_28_S3 ,
         CM_ALM        := "dbPlcHmiALM".ALM[10359] ,
       );

NETWORK
TITLE = 10360 - LCP112_N621_BP1626 - Zone 6 Circulation Fan  - Diff. Pressure Circ. Fan 6

       CALL #"LCP112_N621_BP1626"
       (
         CM_No       := 10360 ,
         Tab       := 28 ,
         SubTab       := 8 ,
         CfgType       := 0 ,
         CfgInvert       := True ,
         InputRaw       := LCP112_N621_BP1626_DI_Ps ,
         SC_Local       := SL_28_S3 ,
         CM_ALM        := "dbPlcHmiALM".ALM[10360] ,
       );

NETWORK
TITLE = 10361 - LCP112_ES01_SF6661 - Emergency Stop  - Dryer 3 Zone 6Area

       CALL #"LCP112_ES01_SF6661"
       (
         CM_No       := 10361 ,
         Tab       := 1 ,
         SubTab       := 6 ,
         CfgType       := 0 ,
         CfgInvert       := True ,
         InputRaw       := LCP112_ES01_SF6661_DI_ChA ,
         SC_Local       := SL_01 ,
         CM_ALM        := "dbPlcHmiALM".ALM[10361] ,
       );

NETWORK
TITLE = 10362 - LCP112_ES01_SF6662 - Emergency Stop  - LCP112

       CALL #"LCP112_ES01_SF6662"
       (
         CM_No       := 10362 ,
         Tab       := 1 ,
         SubTab       := 6 ,
         CfgType       := 0 ,
         CfgInvert       := True ,
         InputRaw       := LCP112_ES01_SF6662_DI_ChA ,
         SC_Local       := SL_01 ,
         CM_ALM        := "dbPlcHmiALM".ALM[10362] ,
       );

NETWORK
TITLE = 10363 - LCP112_DC01_FC1000 - Power Feed Module 24VDC - Status

       CALL #"LCP112_DC01_FC1000"
       (
         CM_No       := 10363 ,
         Tab       := 13 ,
         SubTab       := 6 ,
         CfgType       := 0 ,
         CfgInvert       := True ,
         InputRaw       := LCP112_DC01_FC1000_DI_Flt ,
         SC_Local       := SL_13 ,
         CM_ALM        := "dbPlcHmiALM".ALM[10363] ,
       );

NETWORK
TITLE = 10364 - LCP112_IO_KF1000 - Point IO - EtherNet/IP Adapter

       CALL #"LCP112_IO_KF1000"
       (
         CM_No       := 10364 ,
         Tab       := 13 ,
         SubTab       := 6 ,
         CfgType       := 0 ,
         CfgInvert       := True ,
         InputRaw       :=  ,
         SC_Local       := SL_13 ,
         CM_ALM        := "dbPlcHmiALM".ALM[10364] ,
       );

NETWORK
TITLE = 10365 - LCP112_IO_KF3013 - 24V DC 8-Point Safety Input Module - SDI

       CALL #"LCP112_IO_KF3013"
       (
         CM_No       := 10365 ,
         Tab       := 13 ,
         SubTab       := 6 ,
         CfgType       := 0 ,
         CfgInvert       := True ,
         InputRaw       :=  ,
         SC_Local       := SL_13 ,
         CM_ALM        := "dbPlcHmiALM".ALM[10365] ,
       );

NETWORK
TITLE = 10366 - LCP112_IO_KF3014 - 24V DC 8-Point Safety Input Module - SDI

       CALL #"LCP112_IO_KF3014"
       (
         CM_No       := 10366 ,
         Tab       := 13 ,
         SubTab       := 6 ,
         CfgType       := 0 ,
         CfgInvert       := True ,
         InputRaw       :=  ,
         SC_Local       := SL_13 ,
         CM_ALM        := "dbPlcHmiALM".ALM[10366] ,
       );

NETWORK
TITLE = 10367 - LCP113_AC01_FC3701 - 115VAC Power Supply - Thermal Fault

       CALL #"LCP113_AC01_FC3701"
       (
         CM_No       := 10367 ,
         Tab       := 13 ,
         SubTab       := 6 ,
         CfgType       := 0 ,
         CfgInvert       := True ,
         InputRaw       := LCP113_AC01_FC3701_DI_Flt ,
         SC_Local       := SL_13 ,
         CM_ALM        := "dbPlcHmiALM".ALM[10367] ,
       );

NETWORK
TITLE = 10368 - LCP113_I670_QA1701 - Min Gas Pressure Switch - (-BP8701)

       CALL #"LCP113_I670_QA1701"
       (
         CM_No       := 10368 ,
         Tab       := 28 ,
         SubTab       := 9 ,
         CfgType       := 0 ,
         CfgInvert       := True ,
         InputRaw       := LCP113_I670_QA1701_DI_FltL ,
         SC_Local       := SL_28_S3 ,
         CM_ALM        := "dbPlcHmiALM".ALM[10368] ,
       );

NETWORK
TITLE = 10369 - LCP113_I670_QA1702 - Max Gas Pressure Switch - (-BP8702)

       CALL #"LCP113_I670_QA1702"
       (
         CM_No       := 10369 ,
         Tab       := 28 ,
         SubTab       := 9 ,
         CfgType       := 0 ,
         CfgInvert       := True ,
         InputRaw       := LCP113_I670_QA1702_DI_FltH ,
         SC_Local       := SL_28_S3 ,
         CM_ALM        := "dbPlcHmiALM".ALM[10369] ,
       );

NETWORK
TITLE = 10370 - LCP113_I670_QA1703 - Leak Gas Pressure Switch - (-BP8703)

       CALL #"LCP113_I670_QA1703"
       (
         CM_No       := 10370 ,
         Tab       := 28 ,
         SubTab       := 9 ,
         CfgType       := 0 ,
         CfgInvert       := True ,
         InputRaw       := LCP113_I670_QA1703_DI_Ps ,
         SC_Local       := SL_28_S3 ,
         CM_ALM        := "dbPlcHmiALM".ALM[10370] ,
       );

NETWORK
TITLE = 10371 - LCP113_I670_QA1713 - No Air Check Pressure Switch - (-BP2713)

       CALL #"LCP113_I670_QA1713"
       (
         CM_No       := 10371 ,
         Tab       := 28 ,
         SubTab       := 9 ,
         CfgType       := 0 ,
         CfgInvert       := True ,
         InputRaw       := LCP113_I670_QA1713_DI_Ps ,
         SC_Local       := SL_28_S3 ,
         CM_ALM        := "dbPlcHmiALM".ALM[10371] ,
       );

NETWORK
TITLE = 10372 - LCP113_I670_QA1708 - Burner Failure - Signal from Maxon

       CALL #"LCP113_I670_QA1708"
       (
         CM_No       := 10372 ,
         Tab       := 28 ,
         SubTab       := 9 ,
         CfgType       := 0 ,
         CfgInvert       := True ,
         InputRaw       := LCP113_I670_QA1708_DI_Flt ,
         SC_Local       := SL_28_S3 ,
         CM_ALM        := "dbPlcHmiALM".ALM[10372] ,
       );

NETWORK
TITLE = 10373 - LCP113_I670_QA1704 - High Temperature Failure - Signal from JUMO

       CALL #"LCP113_I670_QA1704"
       (
         CM_No       := 10373 ,
         Tab       := 28 ,
         SubTab       := 9 ,
         CfgType       := 0 ,
         CfgInvert       := True ,
         InputRaw       := LCP113_I670_QA1704_DI_Flt ,
         SC_Local       := SL_28_S3 ,
         CM_ALM        := "dbPlcHmiALM".ALM[10373] ,
       );

NETWORK
TITLE = 10374 - LCP113_N532_BG7701 - Disc Filter 7 Door 1 - Before Filter

       CALL #"LCP113_N532_BG7701"
       (
         CM_No       := 10374 ,
         Tab       := 1 ,
         SubTab       := 8 ,
         CfgType       := 0 ,
         CfgInvert       := True ,
         InputRaw       := LCP113_N532_BG7701_DI_ChA ,
         SC_Local       := SL_28_S3 ,
         CM_ALM        := "dbPlcHmiALM".ALM[10374] ,
       );

NETWORK
TITLE = 10375 - LCP113_N532_BG7703 - Disc Filter 7 Door 2 - After Filter

       CALL #"LCP113_N532_BG7703"
       (
         CM_No       := 10375 ,
         Tab       := 1 ,
         SubTab       := 8 ,
         CfgType       := 0 ,
         CfgInvert       := True ,
         InputRaw       := LCP113_N532_BG7703_DI_ChA ,
         SC_Local       := SL_28_S3 ,
         CM_ALM        := "dbPlcHmiALM".ALM[10375] ,
       );

NETWORK
TITLE = 10376 - LCP113_N631_BP1727 - Zone 7 Circulation Fan - Diff. Pressure Circ. Fan 7

       CALL #"LCP113_N631_BP1727"
       (
         CM_No       := 10376 ,
         Tab       := 28 ,
         SubTab       := 9 ,
         CfgType       := 0 ,
         CfgInvert       := True ,
         InputRaw       := LCP113_N631_BP1727_DI_Ps ,
         SC_Local       := SL_28_S3 ,
         CM_ALM        := "dbPlcHmiALM".ALM[10376] ,
       );

NETWORK
TITLE = 10377 - LCP113_ES01_SF6762 - Emergency Stop  - Dryer 3 Zone 7 Area

       CALL #"LCP113_ES01_SF6762"
       (
         CM_No       := 10377 ,
         Tab       := 1 ,
         SubTab       := 6 ,
         CfgType       := 0 ,
         CfgInvert       := True ,
         InputRaw       := LCP113_ES01_SF6762_DI_ChA ,
         SC_Local       := SL_01 ,
         CM_ALM        := "dbPlcHmiALM".ALM[10377] ,
       );

NETWORK
TITLE = 10378 - LCP113_ES01_SF6763 - Emergency Stop  - LCP113

       CALL #"LCP113_ES01_SF6763"
       (
         CM_No       := 10378 ,
         Tab       := 1 ,
         SubTab       := 6 ,
         CfgType       := 0 ,
         CfgInvert       := True ,
         InputRaw       := LCP113_ES01_SF6763_DI_ChA ,
         SC_Local       := SL_01 ,
         CM_ALM        := "dbPlcHmiALM".ALM[10378] ,
       );

NETWORK
TITLE = 10379 - LCP113_DC01_FC1000 - Power Feed Module 24VDC - Status

       CALL #"LCP113_DC01_FC1000"
       (
         CM_No       := 10379 ,
         Tab       := 13 ,
         SubTab       := 6 ,
         CfgType       := 0 ,
         CfgInvert       := True ,
         InputRaw       := LCP113_DC01_FC1000_DI_Flt ,
         SC_Local       := SL_13 ,
         CM_ALM        := "dbPlcHmiALM".ALM[10379] ,
       );

NETWORK
TITLE = 10380 - LCP113_IO_KF1000 - Point IO - EtherNet/IP Adapter

       CALL #"LCP113_IO_KF1000"
       (
         CM_No       := 10380 ,
         Tab       := 13 ,
         SubTab       := 6 ,
         CfgType       := 0 ,
         CfgInvert       := True ,
         InputRaw       :=  ,
         SC_Local       := SL_13 ,
         CM_ALM        := "dbPlcHmiALM".ALM[10380] ,
       );

NETWORK
TITLE = 10381 - LCP113_IO_KF3013 - 24V DC 8-Point Safety Input Module - SDI

       CALL #"LCP113_IO_KF3013"
       (
         CM_No       := 10381 ,
         Tab       := 13 ,
         SubTab       := 6 ,
         CfgType       := 0 ,
         CfgInvert       := True ,
         InputRaw       :=  ,
         SC_Local       := SL_13 ,
         CM_ALM        := "dbPlcHmiALM".ALM[10381] ,
       );

NETWORK
TITLE = 10382 - LCP113_IO_KF3014 - 24V DC 8-Point Safety Input Module - SDI

       CALL #"LCP113_IO_KF3014"
       (
         CM_No       := 10382 ,
         Tab       := 13 ,
         SubTab       := 6 ,
         CfgType       := 0 ,
         CfgInvert       := True ,
         InputRaw       :=  ,
         SC_Local       := SL_13 ,
         CM_ALM        := "dbPlcHmiALM".ALM[10382] ,
       );

NETWORK
TITLE = 10383 - LCP121_ES01_SF6181 - Emergency Stop  - CB.121-01

       CALL #"LCP121_ES01_SF6181"
       (
         CM_No       := 10383 ,
         Tab       := 1 ,
         SubTab       := 7 ,
         CfgType       := 0 ,
         CfgInvert       := True ,
         InputRaw       := LCP121_ES01_SF6181_DI_ChA ,
         SC_Local       := SL_01 ,
         CM_ALM        := "dbPlcHmiALM".ALM[10383] ,
       );

NETWORK
TITLE = 10384 - LCP121_ES01_SF6182 - Emergency Stop  - CB.121-02

       CALL #"LCP121_ES01_SF6182"
       (
         CM_No       := 10384 ,
         Tab       := 1 ,
         SubTab       := 7 ,
         CfgType       := 0 ,
         CfgInvert       := True ,
         InputRaw       := LCP121_ES01_SF6182_DI_ChA ,
         SC_Local       := SL_01 ,
         CM_ALM        := "dbPlcHmiALM".ALM[10384] ,
       );

NETWORK
TITLE = 10385 - LCP121_DC01_FC1000 - Power Feed Module 24VDC - Status

       CALL #"LCP121_DC01_FC1000"
       (
         CM_No       := 10385 ,
         Tab       := 13 ,
         SubTab       := 7 ,
         CfgType       := 0 ,
         CfgInvert       := True ,
         InputRaw       := LCP121_DC01_FC1000_DI_Flt ,
         SC_Local       := SL_13 ,
         CM_ALM        := "dbPlcHmiALM".ALM[10385] ,
       );

NETWORK
TITLE = 10386 - LCP122_ES01_SF6184 - Emergency Stop  - CB122-01

       CALL #"LCP122_ES01_SF6184"
       (
         CM_No       := 10386 ,
         Tab       := 1 ,
         SubTab       := 7 ,
         CfgType       := 0 ,
         CfgInvert       := True ,
         InputRaw       := LCP122_ES01_SF6184_DI_ChA ,
         SC_Local       := SL_01 ,
         CM_ALM        := "dbPlcHmiALM".ALM[10386] ,
       );

NETWORK
TITLE = 10387 - LCP122_ES01_SF6185 - Emergency Stop  - CB122-02

       CALL #"LCP122_ES01_SF6185"
       (
         CM_No       := 10387 ,
         Tab       := 1 ,
         SubTab       := 7 ,
         CfgType       := 0 ,
         CfgInvert       := True ,
         InputRaw       := LCP122_ES01_SF6185_DI_ChA ,
         SC_Local       := SL_01 ,
         CM_ALM        := "dbPlcHmiALM".ALM[10387] ,
       );

NETWORK
TITLE = 10388 - LCP122_ES01_SF6186 - Emergency Stop  - CB.122-03

       CALL #"LCP122_ES01_SF6186"
       (
         CM_No       := 10388 ,
         Tab       := 1 ,
         SubTab       := 7 ,
         CfgType       := 0 ,
         CfgInvert       := True ,
         InputRaw       := LCP122_ES01_SF6186_DI_ChA ,
         SC_Local       := SL_01 ,
         CM_ALM        := "dbPlcHmiALM".ALM[10388] ,
       );

NETWORK
TITLE = 10389 - LCP122_DC01_FC1000 - Power Feed Module 24VDC - Status

       CALL #"LCP122_DC01_FC1000"
       (
         CM_No       := 10389 ,
         Tab       := 13 ,
         SubTab       := 7 ,
         CfgType       := 0 ,
         CfgInvert       := True ,
         InputRaw       := LCP122_DC01_FC1000_DI_Flt ,
         SC_Local       := SL_13 ,
         CM_ALM        := "dbPlcHmiALM".ALM[10389] ,
       );

NETWORK
TITLE = 10390 - LCP123_ES01_SF6188 - Emergency Stop  - CB.123-01

       CALL #"LCP123_ES01_SF6188"
       (
         CM_No       := 10390 ,
         Tab       := 1 ,
         SubTab       := 7 ,
         CfgType       := 0 ,
         CfgInvert       := True ,
         InputRaw       := LCP123_ES01_SF6188_DI_ChA ,
         SC_Local       := SL_01 ,
         CM_ALM        := "dbPlcHmiALM".ALM[10390] ,
       );

NETWORK
TITLE = 10391 - LCP122_ES01_SF6190 - Emergency Stop  - CB.122-04

       CALL #"LCP122_ES01_SF6190"
       (
         CM_No       := 10391 ,
         Tab       := 1 ,
         SubTab       := 7 ,
         CfgType       := 0 ,
         CfgInvert       := True ,
         InputRaw       := LCP122_ES01_SF6190_DI_ChA ,
         SC_Local       := SL_01 ,
         CM_ALM        := "dbPlcHmiALM".ALM[10391] ,
       );

NETWORK
TITLE = 10392 - LCP123_DC01_FC1000 - Power Feed Module 24VDC - Status

       CALL #"LCP123_DC01_FC1000"
       (
         CM_No       := 10392 ,
         Tab       := 13 ,
         SubTab       := 7 ,
         CfgType       := 0 ,
         CfgInvert       := True ,
         InputRaw       := LCP123_DC01_FC1000_DI_Flt ,
         SC_Local       := SL_13 ,
         CM_ALM        := "dbPlcHmiALM".ALM[10392] ,
       );

NETWORK
TITLE = 10393 - LCP121_IO_KF1000 - Point IO - EtherNet/IP Adapter

       CALL #"LCP121_IO_KF1000"
       (
         CM_No       := 10393 ,
         Tab       := 13 ,
         SubTab       := 5 ,
         CfgType       := 0 ,
         CfgInvert       := True ,
         InputRaw       :=  ,
         SC_Local       := SL_13 ,
         CM_ALM        := "dbPlcHmiALM".ALM[10393] ,
       );

NETWORK
TITLE = 10394 - LCP121_IO_KF3010 - 24V DC 8-Point Safety Input Module - SDI

       CALL #"LCP121_IO_KF3010"
       (
         CM_No       := 10394 ,
         Tab       := 13 ,
         SubTab       := 5 ,
         CfgType       := 0 ,
         CfgInvert       := True ,
         InputRaw       :=  ,
         SC_Local       := SL_13 ,
         CM_ALM        := "dbPlcHmiALM".ALM[10394] ,
       );

NETWORK
TITLE = 10395 - LCP131_I811_BP1201 - Zone 1 Burner Fan - Differential Pressure Sensor

       CALL #"LCP131_I811_BP1201"
       (
         CM_No       := 10395 ,
         Tab       := 28 ,
         SubTab       := 3 ,
         CfgType       := 0 ,
         CfgInvert       := True ,
         InputRaw       := LCP131_I811_BP1201_DI_Ps ,
         SC_Local       := SL_28_S1 ,
         CM_ALM        := "dbPlcHmiALM".ALM[10395] ,
       );

NETWORK
TITLE = 10396 - LCP131_K811_BP1202 - Zone 3 Burner Fan - Differential Pressure Sensor

       CALL #"LCP131_K811_BP1202"
       (
         CM_No       := 10396 ,
         Tab       := 28 ,
         SubTab       := 5 ,
         CfgType       := 0 ,
         CfgInvert       := True ,
         InputRaw       := LCP131_K811_BP1202_DI_Ps ,
         SC_Local       := SL_28_S2 ,
         CM_ALM        := "dbPlcHmiALM".ALM[10396] ,
       );

NETWORK
TITLE = 10397 - LCP131_K821_BP1203 - Zone 4 Burner Fan - Differential Pressure Sensor

       CALL #"LCP131_K821_BP1203"
       (
         CM_No       := 10397 ,
         Tab       := 28 ,
         SubTab       := 6 ,
         CfgType       := 0 ,
         CfgInvert       := True ,
         InputRaw       := LCP131_K821_BP1203_DI_Ps ,
         SC_Local       := SL_28_S2 ,
         CM_ALM        := "dbPlcHmiALM".ALM[10397] ,
       );

NETWORK
TITLE = 10398 - LCP131_N811_BP1204 - Zone 5 Burner Fan - Differential Pressure Sensor

       CALL #"LCP131_N811_BP1204"
       (
         CM_No       := 10398 ,
         Tab       := 28 ,
         SubTab       := 7 ,
         CfgType       := 0 ,
         CfgInvert       := True ,
         InputRaw       := LCP131_N811_BP1204_DI_Ps ,
         SC_Local       := SL_28_S3 ,
         CM_ALM        := "dbPlcHmiALM".ALM[10398] ,
       );

NETWORK
TITLE = 10399 - LCP131_N821_BP1205 - Zone 6 Burner Fan - Differential Pressure Sensor

       CALL #"LCP131_N821_BP1205"
       (
         CM_No       := 10399 ,
         Tab       := 28 ,
         SubTab       := 8 ,
         CfgType       := 0 ,
         CfgInvert       := True ,
         InputRaw       := LCP131_N821_BP1205_DI_Ps ,
         SC_Local       := SL_28_S3 ,
         CM_ALM        := "dbPlcHmiALM".ALM[10399] ,
       );

NETWORK
TITLE = 10400 - LCP131_N831_BP1206 - Zone 7 Burner Fan - Differential Pressure Sensor

       CALL #"LCP131_N831_BP1206"
       (
         CM_No       := 10400 ,
         Tab       := 28 ,
         SubTab       := 9 ,
         CfgType       := 0 ,
         CfgInvert       := True ,
         InputRaw       := LCP131_N831_BP1206_DI_Ps ,
         SC_Local       := SL_28_S3 ,
         CM_ALM        := "dbPlcHmiALM".ALM[10400] ,
       );

NETWORK
TITLE = 10401 - LCP131_I711_BP1207 - Exhaust Fan 1 - Differential Pressure Sensor

       CALL #"LCP131_I711_BP1207"
       (
         CM_No       := 10401 ,
         Tab       := 28 ,
         SubTab       := 3 ,
         CfgType       := 0 ,
         CfgInvert       := True ,
         InputRaw       := LCP131_I711_BP1207_DI_Ps ,
         SC_Local       := SL_28_S1 ,
         CM_ALM        := "dbPlcHmiALM".ALM[10401] ,
       );

NETWORK
TITLE = 10402 - LCP131_K711_BP1208 - Exhaust Fan 3 - Differential Pressure Sensor

       CALL #"LCP131_K711_BP1208"
       (
         CM_No       := 10402 ,
         Tab       := 28 ,
         SubTab       := 5 ,
         CfgType       := 0 ,
         CfgInvert       := True ,
         InputRaw       := LCP131_K711_BP1208_DI_Ps ,
         SC_Local       := SL_28_S2 ,
         CM_ALM        := "dbPlcHmiALM".ALM[10402] ,
       );

NETWORK
TITLE = 10403 - LCP131_K721_BP1209 - Exhaust Fan 4 - Differential Pressure Sensor

       CALL #"LCP131_K721_BP1209"
       (
         CM_No       := 10403 ,
         Tab       := 28 ,
         SubTab       := 6 ,
         CfgType       := 0 ,
         CfgInvert       := True ,
         InputRaw       := LCP131_K721_BP1209_DI_Ps ,
         SC_Local       := SL_28_S2 ,
         CM_ALM        := "dbPlcHmiALM".ALM[10403] ,
       );

NETWORK
TITLE = 10404 - LCP131_N711_BP1210 - Exhaust Fan 5 - Differential Pressure Sensor

       CALL #"LCP131_N711_BP1210"
       (
         CM_No       := 10404 ,
         Tab       := 28 ,
         SubTab       := 7 ,
         CfgType       := 0 ,
         CfgInvert       := True ,
         InputRaw       := LCP131_N711_BP1210_DI_Ps ,
         SC_Local       := SL_28_S3 ,
         CM_ALM        := "dbPlcHmiALM".ALM[10404] ,
       );

NETWORK
TITLE = 10405 - LCP131_N721_BP1211 - Exhaust Fan 6 - Differential Pressure Sensor

       CALL #"LCP131_N721_BP1211"
       (
         CM_No       := 10405 ,
         Tab       := 28 ,
         SubTab       := 8 ,
         CfgType       := 0 ,
         CfgInvert       := True ,
         InputRaw       := LCP131_N721_BP1211_DI_Ps ,
         SC_Local       := SL_28_S3 ,
         CM_ALM        := "dbPlcHmiALM".ALM[10405] ,
       );

NETWORK
TITLE = 10406 - LCP131_N731_BP1212 - Exhaust Fan 7 - Differential Pressure Sensor

       CALL #"LCP131_N731_BP1212"
       (
         CM_No       := 10406 ,
         Tab       := 28 ,
         SubTab       := 9 ,
         CfgType       := 0 ,
         CfgInvert       := True ,
         InputRaw       := LCP131_N731_BP1212_DI_Ps ,
         SC_Local       := SL_28_S3 ,
         CM_ALM        := "dbPlcHmiALM".ALM[10406] ,
       );

NETWORK
TITLE = 10407 - LCP131_ES01_SF6191 - Emergency Stop  - Fan Area

       CALL #"LCP131_ES01_SF6191"
       (
         CM_No       := 10407 ,
         Tab       := 1 ,
         SubTab       := 6 ,
         CfgType       := 0 ,
         CfgInvert       := True ,
         InputRaw       := LCP131_ES01_SF6191_DI_ChA ,
         SC_Local       := SL_01 ,
         CM_ALM        := "dbPlcHmiALM".ALM[10407] ,
       );

NETWORK
TITLE = 10408 - LCP131_ES01_SF6192 - Emergency Stop  - Fan Area

